   1:  PR[91,1] = PR[90,1] + 5.124;
   1:  PR[91,2] = PR[90,2] + -25.646;
   1:L PR[91] R[100]mm/sec CNT100;
   1:  PR[91,1] = PR[90,1] + 6.998;
   1:  PR[91,2] = PR[90,2] + -25.330;
   1:L PR[91] R[100]mm/sec CNT100;
   1:  PR[91,1] = PR[90,1] + 9.946;
   1:  PR[91,2] = PR[90,2] + -24.476;
   1:L PR[91] R[100]mm/sec CNT100;
   1:  PR[91,1] = PR[90,1] + 11.813;
   1:  PR[91,2] = PR[90,2] + -23.728;
   1:L PR[91] R[100]mm/sec CNT100;
   1:  PR[91,1] = PR[90,1] + 14.404;
   1:  PR[91,2] = PR[90,2] + -22.433;
   1:L PR[91] R[100]mm/sec CNT100;
   1:  PR[91,1] = PR[90,1] + 16.150;
   1:  PR[91,2] = PR[90,2] + -21.252;
   1:L PR[91] R[100]mm/sec CNT100;
   1:  PR[91,1] = PR[90,1] + 18.488;
   1:  PR[91,2] = PR[90,2] + -19.489;
   1:L PR[91] R[100]mm/sec CNT100;
   1:  PR[91,1] = PR[90,1] + 19.988;
   1:  PR[91,2] = PR[90,2] + -17.914;
   1:L PR[91] R[100]mm/sec CNT100;
   1:  PR[91,1] = PR[90,1] + 22.105;
   1:  PR[91,2] = PR[90,2] + -15.542;
   1:L PR[91] R[100]mm/sec CNT100;
   1:  PR[91,1] = PR[90,1] + 23.235;
   1:  PR[91,2] = PR[90,2] + -13.678;
   1:L PR[91] R[100]mm/sec CNT100;
   1:  PR[91,1] = PR[90,1] + 24.761;
   1:  PR[91,2] = PR[90,2] + -11.061;
   1:L PR[91] R[100]mm/sec CNT100;
   1:  PR[91,1] = PR[90,1] + 25.483;
   1:  PR[91,2] = PR[90,2] + -8.945;
   1:L PR[91] R[100]mm/sec CNT100;
   1:  PR[91,1] = PR[90,1] + 26.090;
   1:  PR[91,2] = PR[90,2] + -7.419;
   1:L PR[91] R[100]mm/sec CNT100;
   1:  PR[91,1] = PR[90,1] + 26.501;
   1:  PR[91,2] = PR[90,2] + -5.955;
   1:L PR[91] R[100]mm/sec CNT100;
   1:  PR[91,1] = PR[90,1] + 26.770;
   1:  PR[91,2] = PR[90,2] + -4.345;
   1:L PR[91] R[100]mm/sec CNT100;
   1:  PR[91,1] = PR[90,1] + 27.018;
   1:  PR[91,2] = PR[90,2] + -2.078;
   1:L PR[91] R[100]mm/sec CNT100;
   1:  PR[91,1] = PR[90,1] + 27.107;
   1:  PR[91,2] = PR[90,2] + -0.484;
   1:L PR[91] R[100]mm/sec CNT100;
   1:  PR[91,1] = PR[90,1] + 26.536;
   1:  PR[91,2] = PR[90,2] + 4.905;
   1:L PR[91] R[100]mm/sec CNT100;
   1:  PR[91,1] = PR[90,1] + 25.602;
   1:  PR[91,2] = PR[90,2] + 7.850;
   1:L PR[91] R[100]mm/sec CNT100;
   1:  PR[91,1] = PR[90,1] + 24.902;
   1:  PR[91,2] = PR[90,2] + 9.901;
   1:L PR[91] R[100]mm/sec CNT100;
   1:  PR[91,1] = PR[90,1] + 23.362;
   1:  PR[91,2] = PR[90,2] + 12.656;
   1:L PR[91] R[100]mm/sec CNT100;
   1:  PR[91,1] = PR[90,1] + 22.206;
   1:  PR[91,2] = PR[90,2] + 14.563;
   1:L PR[91] R[100]mm/sec CNT100;
   1:  PR[91,1] = PR[90,1] + 21.245;
   1:  PR[91,2] = PR[90,2] + 15.786;
   1:L PR[91] R[100]mm/sec CNT100;
   1:  PR[91,1] = PR[90,1] + 19.705;
   1:  PR[91,2] = PR[90,2] + 17.404;
   1:L PR[91] R[100]mm/sec CNT100;
   1:  PR[91,1] = PR[90,1] + 18.475;
   1:  PR[91,2] = PR[90,2] + 18.659;
   1:L PR[91] R[100]mm/sec CNT100;
   1:  PR[91,1] = PR[90,1] + 17.022;
   1:  PR[91,2] = PR[90,2] + 19.828;
   1:L PR[91] R[100]mm/sec CNT100;
   1:  PR[91,1] = PR[90,1] + 15.212;
   1:  PR[91,2] = PR[90,2] + 21.053;
   1:L PR[91] R[100]mm/sec CNT100;
   1:  PR[91,1] = PR[90,1] + 13.555;
   1:  PR[91,2] = PR[90,2] + 22.079;
   1:L PR[91] R[100]mm/sec CNT100;
   1:  PR[91,1] = PR[90,1] + 11.797;
   1:  PR[91,2] = PR[90,2] + 22.888;
   1:L PR[91] R[100]mm/sec CNT100;
   1:  PR[91,1] = PR[90,1] + 9.812;
   1:  PR[91,2] = PR[90,2] + 23.683;
   1:L PR[91] R[100]mm/sec CNT100;
   1:  PR[91,1] = PR[90,1] + 7.974;
   1:  PR[91,2] = PR[90,2] + 24.268;
   1:L PR[91] R[100]mm/sec CNT100;
   1:  PR[91,1] = PR[90,1] + 5.960;
   1:  PR[91,2] = PR[90,2] + 24.606;
   1:L PR[91] R[100]mm/sec CNT100;
   1:  PR[91,1] = PR[90,1] + 3.894;
   1:  PR[91,2] = PR[90,2] + 24.993;
   1:L PR[91] R[100]mm/sec CNT100;
   1:  PR[91,1] = PR[90,1] + 1.941;
   1:  PR[91,2] = PR[90,2] + 25.113;
   1:L PR[91] R[100]mm/sec CNT100;
   1:  PR[91,1] = PR[90,1] + -0.146;
   1:  PR[91,2] = PR[90,2] + 25.027;
   1:L PR[91] R[100]mm/sec CNT100;
   1:  PR[91] = PR[90];
   1:  PR[91,1] = PR[90,1] + -1.780;
   1:  PR[91,2] = PR[90,2] + 25.420;
   1:  PR[91,3] = PR[90,3] + 71.695;
   1:L PR[91] R[100]mm/sec CNT100;
   1:  PR[91,1] = PR[90,1] + -4.146;
   1:  PR[91,2] = PR[90,2] + 25.274;
   1:L PR[91] R[100]mm/sec CNT100;
   1:  PR[91,1] = PR[90,1] + -5.565;
   1:  PR[91,2] = PR[90,2] + 25.035;
   1:L PR[91] R[100]mm/sec CNT100;
   1:  PR[91,1] = PR[90,1] + -7.940;
   1:  PR[91,2] = PR[90,2] + 24.591;
   1:L PR[91] R[100]mm/sec CNT100;
   1:  PR[91,1] = PR[90,1] + -10.180;
   1:  PR[91,2] = PR[90,2] + 23.878;
   1:L PR[91] R[100]mm/sec CNT100;
   1:  PR[91,1] = PR[90,1] + -11.552;
   1:  PR[91,2] = PR[90,2] + 23.329;
   1:L PR[91] R[100]mm/sec CNT100;
   1:  PR[91,1] = PR[90,1] + -13.642;
   1:  PR[91,2] = PR[90,2] + 22.367;
   1:L PR[91] R[100]mm/sec CNT100;
   1:  PR[91,1] = PR[90,1] + -14.917;
   1:  PR[91,2] = PR[90,2] + 21.506;
   1:L PR[91] R[100]mm/sec CNT100;
   1:  PR[91,1] = PR[90,1] + -16.981;
   1:  PR[91,2] = PR[90,2] + 20.227;
   1:L PR[91] R[100]mm/sec CNT100;
   1:  PR[91,1] = PR[90,1] + -18.712;
   1:  PR[91,2] = PR[90,2] + 18.833;
   1:L PR[91] R[100]mm/sec CNT100;
   1:  PR[91,1] = PR[90,1] + -19.758;
   1:  PR[91,2] = PR[90,2] + 17.736;
   1:L PR[91] R[100]mm/sec CNT100;
   1:  PR[91,1] = PR[90,1] + -22.355;
   1:  PR[91,2] = PR[90,2] + 14.827;
   1:L PR[91] R[100]mm/sec CNT100;
   1:  PR[91,1] = PR[90,1] + -23.115;
   1:  PR[91,2] = PR[90,2] + 13.573;
   1:L PR[91] R[100]mm/sec CNT100;
   1:  PR[91,1] = PR[90,1] + -24.999;
   1:  PR[91,2] = PR[90,2] + 10.343;
   1:L PR[91] R[100]mm/sec CNT100;
   1:  PR[91,1] = PR[90,1] + -25.488;
   1:  PR[91,2] = PR[90,2] + 8.909;
   1:L PR[91] R[100]mm/sec CNT100;
   1:  PR[91,1] = PR[90,1] + -26.233;
   1:  PR[91,2] = PR[90,2] + 7.034;
   1:L PR[91] R[100]mm/sec CNT100;
   1:  PR[91,1] = PR[90,1] + -26.751;
   1:  PR[91,2] = PR[90,2] + 5.192;
   1:L PR[91] R[100]mm/sec CNT100;
   1:  PR[91,1] = PR[90,1] + -27.087;
   1:  PR[91,2] = PR[90,2] + 3.184;
   1:L PR[91] R[100]mm/sec CNT100;
   1:  PR[91,1] = PR[90,1] + -27.255;
   1:  PR[91,2] = PR[90,2] + 1.644;
   1:L PR[91] R[100]mm/sec CNT100;
   1:  PR[91,1] = PR[90,1] + -27.367;
   1:  PR[91,2] = PR[90,2] + -0.364;
   1:L PR[91] R[100]mm/sec CNT100;
   1:  PR[91,1] = PR[90,1] + -26.796;
   1:  PR[91,2] = PR[90,2] + -5.788;
   1:L PR[91] R[100]mm/sec CNT100;
   1:  PR[91,1] = PR[90,1] + -25.639;
   1:  PR[91,2] = PR[90,2] + -9.436;
   1:L PR[91] R[100]mm/sec CNT100;
   1:  PR[91,1] = PR[90,1] + -25.172;
   1:  PR[91,2] = PR[90,2] + -10.805;
   1:L PR[91] R[100]mm/sec CNT100;
   1:  PR[91,1] = PR[90,1] + -23.273;
   1:  PR[91,2] = PR[90,2] + -14.201;
   1:L PR[91] R[100]mm/sec CNT100;
   1:  PR[91,1] = PR[90,1] + -22.487;
   1:  PR[91,2] = PR[90,2] + -15.498;
   1:L PR[91] R[100]mm/sec CNT100;
   1:  PR[91,1] = PR[90,1] + -21.291;
   1:  PR[91,2] = PR[90,2] + -17.021;
   1:L PR[91] R[100]mm/sec CNT100;
   1:  PR[91,1] = PR[90,1] + -20.228;
   1:  PR[91,2] = PR[90,2] + -18.137;
   1:L PR[91] R[100]mm/sec CNT100;
   1:  PR[91,1] = PR[90,1] + -18.757;
   1:  PR[91,2] = PR[90,2] + -19.638;
   1:L PR[91] R[100]mm/sec CNT100;
   1:  PR[91,1] = PR[90,1] + -15.723;
   1:  PR[91,2] = PR[90,2] + -21.903;
   1:L PR[91] R[100]mm/sec CNT100;
   1:  PR[91,1] = PR[90,1] + -14.553;
   1:  PR[91,2] = PR[90,2] + -22.694;
   1:L PR[91] R[100]mm/sec CNT100;
   1:  PR[91,1] = PR[90,1] + -11.293;
   1:  PR[91,2] = PR[90,2] + -24.274;
   1:L PR[91] R[100]mm/sec CNT100;
   1:  PR[91,1] = PR[90,1] + -10.048;
   1:  PR[91,2] = PR[90,2] + -24.773;
   1:L PR[91] R[100]mm/sec CNT100;
   1:  PR[91,1] = PR[90,1] + -6.562;
   1:  PR[91,2] = PR[90,2] + -25.731;
   1:L PR[91] R[100]mm/sec CNT100;
   1:  PR[91,1] = PR[90,1] + -5.323;
   1:  PR[91,2] = PR[90,2] + -25.940;
   1:L PR[91] R[100]mm/sec CNT100;
   1:  PR[91,1] = PR[90,1] + -1.628;
   1:  PR[91,2] = PR[90,2] + -26.261;
   1:L PR[91] R[100]mm/sec CNT100;
   1:  PR[91,1] = PR[90,1] + -0.309;
   1:  PR[91,2] = PR[90,2] + -26.206;
   1:L PR[91] R[100]mm/sec CNT100;
   1:  PR[91,1] = PR[90,1] + 1.137;
   1:  PR[91,2] = PR[90,2] + -26.261;
   1:L PR[91] R[100]mm/sec CNT100;
   1:  PR[91,1] = PR[90,1] + 5.091;
   1:  PR[91,2] = PR[90,2] + -25.894;
   1:L PR[91] R[100]mm/sec CNT100;
   1:  PR[91,1] = PR[90,1] + 6.320;
   1:  PR[91,2] = PR[90,2] + -25.686;
   1:L PR[91] R[100]mm/sec CNT100;
   1:  PR[91,1] = PR[90,1] + 9.853;
   1:  PR[91,2] = PR[90,2] + -24.664;
   1:L PR[91] R[100]mm/sec CNT100;
   1:  PR[91,1] = PR[90,1] + 11.098;
   1:  PR[91,2] = PR[90,2] + -24.165;
   1:L PR[91] R[100]mm/sec CNT100;
   1:  PR[91,1] = PR[90,1] + 14.232;
   1:  PR[91,2] = PR[90,2] + -22.598;
   1:L PR[91] R[100]mm/sec CNT100;
   1:  PR[91,1] = PR[90,1] + 15.409;
   1:  PR[91,2] = PR[90,2] + -21.802;
   1:L PR[91] R[100]mm/sec CNT100;
   1:  PR[91,1] = PR[90,1] + 18.260;
   1:  PR[91,2] = PR[90,2] + -19.652;
   1:L PR[91] R[100]mm/sec CNT100;
   1:  PR[91,1] = PR[90,1] + 19.279;
   1:  PR[91,2] = PR[90,2] + -18.582;
   1:L PR[91] R[100]mm/sec CNT100;
   1:  PR[91,1] = PR[90,1] + 21.876;
   1:  PR[91,2] = PR[90,2] + -15.672;
   1:L PR[91] R[100]mm/sec CNT100;
   1:  PR[91,1] = PR[90,1] + 22.636;
   1:  PR[91,2] = PR[90,2] + -14.418;
   1:L PR[91] R[100]mm/sec CNT100;
   1:  PR[91,1] = PR[90,1] + 24.520;
   1:  PR[91,2] = PR[90,2] + -11.188;
   1:L PR[91] R[100]mm/sec CNT100;
   1:  PR[91,1] = PR[90,1] + 25.009;
   1:  PR[91,2] = PR[90,2] + -9.755;
   1:L PR[91] R[100]mm/sec CNT100;
   1:  PR[91,1] = PR[90,1] + 25.754;
   1:  PR[91,2] = PR[90,2] + -7.880;
   1:L PR[91] R[100]mm/sec CNT100;
   1:  PR[91,1] = PR[90,1] + 26.271;
   1:  PR[91,2] = PR[90,2] + -6.039;
   1:L PR[91] R[100]mm/sec CNT100;
   1:  PR[91,1] = PR[90,1] + 26.607;
   1:  PR[91,2] = PR[90,2] + -4.032;
   1:L PR[91] R[100]mm/sec CNT100;
   1:  PR[91,1] = PR[90,1] + 26.776;
   1:  PR[91,2] = PR[90,2] + -2.491;
   1:L PR[91] R[100]mm/sec CNT100;
   1:  PR[91,1] = PR[90,1] + 26.887;
   1:  PR[91,2] = PR[90,2] + -0.483;
   1:L PR[91] R[100]mm/sec CNT100;
   1:  PR[91,1] = PR[90,1] + 26.317;
   1:  PR[91,2] = PR[90,2] + 4.939;
   1:L PR[91] R[100]mm/sec CNT100;
   1:  PR[91,1] = PR[90,1] + 25.160;
   1:  PR[91,2] = PR[90,2] + 8.588;
   1:L PR[91] R[100]mm/sec CNT100;
   1:  PR[91,1] = PR[90,1] + 24.693;
   1:  PR[91,2] = PR[90,2] + 9.956;
   1:L PR[91] R[100]mm/sec CNT100;
   1:  PR[91,1] = PR[90,1] + 22.793;
   1:  PR[91,2] = PR[90,2] + 13.354;
   1:L PR[91] R[100]mm/sec CNT100;
   1:  PR[91,1] = PR[90,1] + 22.006;
   1:  PR[91,2] = PR[90,2] + 14.652;
   1:L PR[91] R[100]mm/sec CNT100;
   1:  PR[91,1] = PR[90,1] + 20.811;
   1:  PR[91,2] = PR[90,2] + 16.174;
   1:L PR[91] R[100]mm/sec CNT100;
   1:  PR[91,1] = PR[90,1] + 19.747;
   1:  PR[91,2] = PR[90,2] + 17.291;
   1:L PR[91] R[100]mm/sec CNT100;
   1:  PR[91,1] = PR[90,1] + 18.247;
   1:  PR[91,2] = PR[90,2] + 18.822;
   1:L PR[91] R[100]mm/sec CNT100;
   1:  PR[91,1] = PR[90,1] + 16.464;
   1:  PR[91,2] = PR[90,2] + 20.257;
   1:L PR[91] R[100]mm/sec CNT100;
   1:  PR[91,1] = PR[90,1] + 15.212;
   1:  PR[91,2] = PR[90,2] + 21.104;
   1:L PR[91] R[100]mm/sec CNT100;
   1:  PR[91,1] = PR[90,1] + 13.205;
   1:  PR[91,2] = PR[90,2] + 22.347;
   1:L PR[91] R[100]mm/sec CNT100;
   1:  PR[91,1] = PR[90,1] + 11.072;
   1:  PR[91,2] = PR[90,2] + 23.329;
   1:L PR[91] R[100]mm/sec CNT100;
   1:  PR[91,1] = PR[90,1] + 9.701;
   1:  PR[91,2] = PR[90,2] + 23.878;
   1:L PR[91] R[100]mm/sec CNT100;
   1:  PR[91,1] = PR[90,1] + 7.481;
   1:  PR[91,2] = PR[90,2] + 24.584;
   1:L PR[91] R[100]mm/sec CNT100;
   1:  PR[91,1] = PR[90,1] + 6.092;
   1:  PR[91,2] = PR[90,2] + 24.818;
   1:L PR[91] R[100]mm/sec CNT100;
   1:  PR[91,1] = PR[90,1] + 3.644;
   1:  PR[91,2] = PR[90,2] + 25.275;
   1:L PR[91] R[100]mm/sec CNT100;
   1:  PR[91,1] = PR[90,1] + 1.303;
   1:  PR[91,2] = PR[90,2] + 25.420;
   1:L PR[91] R[100]mm/sec CNT100;
   1:  PR[91,1] = PR[90,1] + -0.172;
   1:  PR[91,2] = PR[90,2] + 25.359;
   1:L PR[91] R[100]mm/sec CNT100;
   1:  PR[91] = PR[90];
   1:  PR[91,1] = PR[90,1] + -1.142;
   1:  PR[91,2] = PR[90,2] + 25.727;
   1:  PR[91,3] = PR[90,3] + 72.995;
   1:L PR[91] R[100]mm/sec CNT100;
   1:  PR[91,1] = PR[90,1] + -3.897;
   1:  PR[91,2] = PR[90,2] + 25.556;
   1:L PR[91] R[100]mm/sec CNT100;
   1:  PR[91,1] = PR[90,1] + -4.679;
   1:  PR[91,2] = PR[90,2] + 25.425;
   1:L PR[91] R[100]mm/sec CNT100;
   1:  PR[91,1] = PR[90,1] + -7.448;
   1:  PR[91,2] = PR[90,2] + 24.907;
   1:L PR[91] R[100]mm/sec CNT100;
   1:  PR[91,1] = PR[90,1] + -10.070;
   1:  PR[91,2] = PR[90,2] + 24.073;
   1:L PR[91] R[100]mm/sec CNT100;
   1:  PR[91,1] = PR[90,1] + -10.827;
   1:  PR[91,2] = PR[90,2] + 23.769;
   1:L PR[91] R[100]mm/sec CNT100;
   1:  PR[91,1] = PR[90,1] + -13.292;
   1:  PR[91,2] = PR[90,2] + 22.635;
   1:L PR[91] R[100]mm/sec CNT100;
   1:  PR[91,1] = PR[90,1] + -13.998;
   1:  PR[91,2] = PR[90,2] + 22.158;
   1:L PR[91] R[100]mm/sec CNT100;
   1:  PR[91,1] = PR[90,1] + -16.423;
   1:  PR[91,2] = PR[90,2] + 20.656;
   1:L PR[91] R[100]mm/sec CNT100;
   1:  PR[91,1] = PR[90,1] + -18.484;
   1:  PR[91,2] = PR[90,2] + 18.996;
   1:L PR[91] R[100]mm/sec CNT100;
   1:  PR[91,1] = PR[90,1] + -19.049;
   1:  PR[91,2] = PR[90,2] + 18.404;
   1:L PR[91] R[100]mm/sec CNT100;
   1:  PR[91,1] = PR[90,1] + -22.125;
   1:  PR[91,2] = PR[90,2] + 14.957;
   1:L PR[91] R[100]mm/sec CNT100;
   1:  PR[91,1] = PR[90,1] + -22.516;
   1:  PR[91,2] = PR[90,2] + 14.313;
   1:L PR[91] R[100]mm/sec CNT100;
   1:  PR[91,1] = PR[90,1] + -24.757;
   1:  PR[91,2] = PR[90,2] + 10.470;
   1:L PR[91] R[100]mm/sec CNT100;
   1:  PR[91,1] = PR[90,1] + -25.013;
   1:  PR[91,2] = PR[90,2] + 9.720;
   1:L PR[91] R[100]mm/sec CNT100;
   1:  PR[91,1] = PR[90,1] + -25.898;
   1:  PR[91,2] = PR[90,2] + 7.495;
   1:L PR[91] R[100]mm/sec CNT100;
   1:  PR[91,1] = PR[90,1] + -26.521;
   1:  PR[91,2] = PR[90,2] + 5.276;
   1:L PR[91] R[100]mm/sec CNT100;
   1:  PR[91,1] = PR[90,1] + -26.923;
   1:  PR[91,2] = PR[90,2] + 2.871;
   1:L PR[91] R[100]mm/sec CNT100;
   1:  PR[91,1] = PR[90,1] + -27.013;
   1:  PR[91,2] = PR[90,2] + 2.056;
   1:L PR[91] R[100]mm/sec CNT100;
   1:  PR[91,1] = PR[90,1] + -27.147;
   1:  PR[91,2] = PR[90,2] + -0.365;
   1:L PR[91] R[100]mm/sec CNT100;
   1:  PR[91,1] = PR[90,1] + -26.577;
   1:  PR[91,2] = PR[90,2] + -5.823;
   1:L PR[91] R[100]mm/sec CNT100;
   1:  PR[91,1] = PR[90,1] + -25.197;
   1:  PR[91,2] = PR[90,2] + -10.174;
   1:L PR[91] R[100]mm/sec CNT100;
   1:  PR[91,1] = PR[90,1] + -24.963;
   1:  PR[91,2] = PR[90,2] + -10.860;
   1:L PR[91] R[100]mm/sec CNT100;
   1:  PR[91,1] = PR[90,1] + -22.704;
   1:  PR[91,2] = PR[90,2] + -14.899;
   1:L PR[91] R[100]mm/sec CNT100;
   1:  PR[91,1] = PR[90,1] + -22.287;
   1:  PR[91,2] = PR[90,2] + -15.587;
   1:L PR[91] R[100]mm/sec CNT100;
   1:  PR[91,1] = PR[90,1] + -20.857;
   1:  PR[91,2] = PR[90,2] + -17.409;
   1:L PR[91] R[100]mm/sec CNT100;
   1:  PR[91,1] = PR[90,1] + -20.271;
   1:  PR[91,2] = PR[90,2] + -18.024;
   1:L PR[91] R[100]mm/sec CNT100;
   1:  PR[91,1] = PR[90,1] + -18.529;
   1:  PR[91,2] = PR[90,2] + -19.802;
   1:L PR[91] R[100]mm/sec CNT100;
   1:  PR[91,1] = PR[90,1] + -14.954;
   1:  PR[91,2] = PR[90,2] + -22.470;
   1:L PR[91] R[100]mm/sec CNT100;
   1:  PR[91,1] = PR[90,1] + -14.353;
   1:  PR[91,2] = PR[90,2] + -22.876;
   1:L PR[91] R[100]mm/sec CNT100;
   1:  PR[91,1] = PR[90,1] + -10.529;
   1:  PR[91,2] = PR[90,2] + -24.729;
   1:L PR[91] R[100]mm/sec CNT100;
   1:  PR[91,1] = PR[90,1] + -9.910;
   1:  PR[91,2] = PR[90,2] + -24.978;
   1:L PR[91] R[100]mm/sec CNT100;
   1:  PR[91,1] = PR[90,1] + -5.845;
   1:  PR[91,2] = PR[90,2] + -26.095;
   1:L PR[91] R[100]mm/sec CNT100;
   1:  PR[91,1] = PR[90,1] + -5.252;
   1:  PR[91,2] = PR[90,2] + -26.195;
   1:L PR[91] R[100]mm/sec CNT100;
   1:  PR[91,1] = PR[90,1] + -0.972;
   1:  PR[91,2] = PR[90,2] + -26.566;
   1:L PR[91] R[100]mm/sec CNT100;
   1:  PR[91,1] = PR[90,1] + -0.283;
   1:  PR[91,2] = PR[90,2] + -26.538;
   1:L PR[91] R[100]mm/sec CNT100;
   1:  PR[91,1] = PR[90,1] + 0.480;
   1:  PR[91,2] = PR[90,2] + -26.567;
   1:L PR[91] R[100]mm/sec CNT100;
   1:  PR[91,1] = PR[90,1] + 5.058;
   1:  PR[91,2] = PR[90,2] + -26.142;
   1:L PR[91] R[100]mm/sec CNT100;
   1:  PR[91,1] = PR[90,1] + 5.643;
   1:  PR[91,2] = PR[90,2] + -26.043;
   1:L PR[91] R[100]mm/sec CNT100;
   1:  PR[91,1] = PR[90,1] + 9.761;
   1:  PR[91,2] = PR[90,2] + -24.851;
   1:L PR[91] R[100]mm/sec CNT100;
   1:  PR[91,1] = PR[90,1] + 10.383;
   1:  PR[91,2] = PR[90,2] + -24.602;
   1:L PR[91] R[100]mm/sec CNT100;
   1:  PR[91,1] = PR[90,1] + 14.059;
   1:  PR[91,2] = PR[90,2] + -22.764;
   1:L PR[91] R[100]mm/sec CNT100;
   1:  PR[91,1] = PR[90,1] + 14.669;
   1:  PR[91,2] = PR[90,2] + -22.351;
   1:L PR[91] R[100]mm/sec CNT100;
   1:  PR[91,1] = PR[90,1] + 18.032;
   1:  PR[91,2] = PR[90,2] + -19.816;
   1:L PR[91] R[100]mm/sec CNT100;
   1:  PR[91,1] = PR[90,1] + 18.570;
   1:  PR[91,2] = PR[90,2] + -19.250;
   1:L PR[91] R[100]mm/sec CNT100;
   1:  PR[91,1] = PR[90,1] + 21.647;
   1:  PR[91,2] = PR[90,2] + -15.803;
   1:L PR[91] R[100]mm/sec CNT100;
   1:  PR[91,1] = PR[90,1] + 22.037;
   1:  PR[91,2] = PR[90,2] + -15.159;
   1:L PR[91] R[100]mm/sec CNT100;
   1:  PR[91,1] = PR[90,1] + 24.279;
   1:  PR[91,2] = PR[90,2] + -11.315;
   1:L PR[91] R[100]mm/sec CNT100;
   1:  PR[91,1] = PR[90,1] + 24.534;
   1:  PR[91,2] = PR[90,2] + -10.566;
   1:L PR[91] R[100]mm/sec CNT100;
   1:  PR[91,1] = PR[90,1] + 25.419;
   1:  PR[91,2] = PR[90,2] + -8.341;
   1:L PR[91] R[100]mm/sec CNT100;
   1:  PR[91,1] = PR[90,1] + 26.041;
   1:  PR[91,2] = PR[90,2] + -6.123;
   1:L PR[91] R[100]mm/sec CNT100;
   1:  PR[91,1] = PR[90,1] + 26.444;
   1:  PR[91,2] = PR[90,2] + -3.718;
   1:L PR[91] R[100]mm/sec CNT100;
   1:  PR[91,1] = PR[90,1] + 26.533;
   1:  PR[91,2] = PR[90,2] + -2.903;
   1:L PR[91] R[100]mm/sec CNT100;
   1:  PR[91,1] = PR[90,1] + 26.668;
   1:  PR[91,2] = PR[90,2] + -0.482;
   1:L PR[91] R[100]mm/sec CNT100;
   1:  PR[91,1] = PR[90,1] + 26.098;
   1:  PR[91,2] = PR[90,2] + 4.972;
   1:L PR[91] R[100]mm/sec CNT100;
   1:  PR[91,1] = PR[90,1] + 24.718;
   1:  PR[91,2] = PR[90,2] + 9.326;
   1:L PR[91] R[100]mm/sec CNT100;
   1:  PR[91,1] = PR[90,1] + 24.484;
   1:  PR[91,2] = PR[90,2] + 10.011;
   1:L PR[91] R[100]mm/sec CNT100;
   1:  PR[91,1] = PR[90,1] + 22.223;
   1:  PR[91,2] = PR[90,2] + 14.053;
   1:L PR[91] R[100]mm/sec CNT100;
   1:  PR[91,1] = PR[90,1] + 21.807;
   1:  PR[91,2] = PR[90,2] + 14.741;
   1:L PR[91] R[100]mm/sec CNT100;
   1:  PR[91,1] = PR[90,1] + 20.376;
   1:  PR[91,2] = PR[90,2] + 16.562;
   1:L PR[91] R[100]mm/sec CNT100;
   1:  PR[91,1] = PR[90,1] + 19.789;
   1:  PR[91,2] = PR[90,2] + 17.179;
   1:L PR[91] R[100]mm/sec CNT100;
   1:  PR[91,1] = PR[90,1] + 18.019;
   1:  PR[91,2] = PR[90,2] + 18.985;
   1:L PR[91] R[100]mm/sec CNT100;
   1:  PR[91,1] = PR[90,1] + 15.906;
   1:  PR[91,2] = PR[90,2] + 20.686;
   1:L PR[91] R[100]mm/sec CNT100;
   1:  PR[91,1] = PR[90,1] + 15.213;
   1:  PR[91,2] = PR[90,2] + 21.155;
   1:L PR[91] R[100]mm/sec CNT100;
   1:  PR[91,1] = PR[90,1] + 12.855;
   1:  PR[91,2] = PR[90,2] + 22.615;
   1:L PR[91] R[100]mm/sec CNT100;
   1:  PR[91,1] = PR[90,1] + 10.347;
   1:  PR[91,2] = PR[90,2] + 23.769;
   1:L PR[91] R[100]mm/sec CNT100;
   1:  PR[91,1] = PR[90,1] + 9.590;
   1:  PR[91,2] = PR[90,2] + 24.073;
   1:L PR[91] R[100]mm/sec CNT100;
   1:  PR[91,1] = PR[90,1] + 6.988;
   1:  PR[91,2] = PR[90,2] + 24.900;
   1:L PR[91] R[100]mm/sec CNT100;
   1:  PR[91,1] = PR[90,1] + 6.224;
   1:  PR[91,2] = PR[90,2] + 25.029;
   1:L PR[91] R[100]mm/sec CNT100;
   1:  PR[91,1] = PR[90,1] + 3.394;
   1:  PR[91,2] = PR[90,2] + 25.558;
   1:L PR[91] R[100]mm/sec CNT100;
   1:  PR[91,1] = PR[90,1] + 0.665;
   1:  PR[91,2] = PR[90,2] + 25.726;
   1:L PR[91] R[100]mm/sec CNT100;
   1:  PR[91,1] = PR[90,1] + -0.199;
   1:  PR[91,2] = PR[90,2] + 25.691;
   1:L PR[91] R[100]mm/sec CNT100;
   1:  PR[91] = PR[90];
   1:  PR[91,1] = PR[90,1] + -0.504;
   1:  PR[91,2] = PR[90,2] + 26.033;
   1:  PR[91,3] = PR[90,3] + 74.295;
   1:L PR[91] R[100]mm/sec CNT100;
   1:  PR[91,1] = PR[90,1] + -3.627;
   1:  PR[91,2] = PR[90,2] + 25.840;
   1:L PR[91] R[100]mm/sec CNT100;
   1:  PR[91,1] = PR[90,1] + -6.957;
   1:  PR[91,2] = PR[90,2] + 25.223;
   1:L PR[91] R[100]mm/sec CNT100;
   1:  PR[91,1] = PR[90,1] + -9.959;
   1:  PR[91,2] = PR[90,2] + 24.267;
   1:L PR[91] R[100]mm/sec CNT100;
   1:  PR[91,1] = PR[90,1] + -10.102;
   1:  PR[91,2] = PR[90,2] + 24.210;
   1:L PR[91] R[100]mm/sec CNT100;
   1:  PR[91,1] = PR[90,1] + -12.942;
   1:  PR[91,2] = PR[90,2] + 22.903;
   1:L PR[91] R[100]mm/sec CNT100;
   1:  PR[91,1] = PR[90,1] + -13.079;
   1:  PR[91,2] = PR[90,2] + 22.810;
   1:L PR[91] R[100]mm/sec CNT100;
   1:  PR[91,1] = PR[90,1] + -15.865;
   1:  PR[91,2] = PR[90,2] + 21.085;
   1:L PR[91] R[100]mm/sec CNT100;
   1:  PR[91,1] = PR[90,1] + -18.227;
   1:  PR[91,2] = PR[90,2] + 19.183;
   1:L PR[91] R[100]mm/sec CNT100;
   1:  PR[91,1] = PR[90,1] + -21.884;
   1:  PR[91,2] = PR[90,2] + 15.100;
   1:L PR[91] R[100]mm/sec CNT100;
   1:  PR[91,1] = PR[90,1] + -24.516;
   1:  PR[91,2] = PR[90,2] + 10.596;
   1:L PR[91] R[100]mm/sec CNT100;
   1:  PR[91,1] = PR[90,1] + -24.538;
   1:  PR[91,2] = PR[90,2] + 10.531;
   1:L PR[91] R[100]mm/sec CNT100;
   1:  PR[91,1] = PR[90,1] + -25.562;
   1:  PR[91,2] = PR[90,2] + 7.957;
   1:L PR[91] R[100]mm/sec CNT100;
   1:  PR[91,1] = PR[90,1] + -26.291;
   1:  PR[91,2] = PR[90,2] + 5.361;
   1:L PR[91] R[100]mm/sec CNT100;
   1:  PR[91,1] = PR[90,1] + -26.760;
   1:  PR[91,2] = PR[90,2] + 2.559;
   1:L PR[91] R[100]mm/sec CNT100;
   1:  PR[91,1] = PR[90,1] + -26.770;
   1:  PR[91,2] = PR[90,2] + 2.469;
   1:L PR[91] R[100]mm/sec CNT100;
   1:  PR[91,1] = PR[90,1] + -26.928;
   1:  PR[91,2] = PR[90,2] + -0.366;
   1:L PR[91] R[100]mm/sec CNT100;
   1:  PR[91,1] = PR[90,1] + -26.358;
   1:  PR[91,2] = PR[90,2] + -5.856;
   1:L PR[91] R[100]mm/sec CNT100;
   1:  PR[91,1] = PR[90,1] + -24.741;
   1:  PR[91,2] = PR[90,2] + -10.937;
   1:L PR[91] R[100]mm/sec CNT100;
   1:  PR[91,1] = PR[90,1] + -22.135;
   1:  PR[91,2] = PR[90,2] + -15.598;
   1:L PR[91] R[100]mm/sec CNT100;
   1:  PR[91,1] = PR[90,1] + -22.088;
   1:  PR[91,2] = PR[90,2] + -15.676;
   1:L PR[91] R[100]mm/sec CNT100;
   1:  PR[91,1] = PR[90,1] + -20.432;
   1:  PR[91,2] = PR[90,2] + -17.784;
   1:L PR[91] R[100]mm/sec CNT100;
   1:  PR[91,1] = PR[90,1] + -18.299;
   1:  PR[91,2] = PR[90,2] + -19.966;
   1:L PR[91] R[100]mm/sec CNT100;
   1:  PR[91,1] = PR[90,1] + -14.185;
   1:  PR[91,2] = PR[90,2] + -23.037;
   1:L PR[91] R[100]mm/sec CNT100;
   1:  PR[91,1] = PR[90,1] + -14.153;
   1:  PR[91,2] = PR[90,2] + -23.058;
   1:L PR[91] R[100]mm/sec CNT100;
   1:  PR[91,1] = PR[90,1] + -9.769;
   1:  PR[91,2] = PR[90,2] + -25.183;
   1:L PR[91] R[100]mm/sec CNT100;
   1:  PR[91,1] = PR[90,1] + -5.151;
   1:  PR[91,2] = PR[90,2] + -26.452;
   1:L PR[91] R[100]mm/sec CNT100;
   1:  PR[91,1] = PR[90,1] + -0.265;
   1:  PR[91,2] = PR[90,2] + -26.877;
   1:L PR[91] R[100]mm/sec CNT100;
   1:  PR[91,1] = PR[90,1] + -0.222;
   1:L PR[91] R[100]mm/sec CNT100;
   1:  PR[91,1] = PR[90,1] + 4.988;
   1:  PR[91,2] = PR[90,2] + -26.393;
   1:L PR[91] R[100]mm/sec CNT100;
   1:  PR[91,1] = PR[90,1] + 9.668;
   1:  PR[91,2] = PR[90,2] + -25.038;
   1:L PR[91] R[100]mm/sec CNT100;
   1:  PR[91,1] = PR[90,1] + 13.887;
   1:  PR[91,2] = PR[90,2] + -22.929;
   1:L PR[91] R[100]mm/sec CNT100;
   1:  PR[91,1] = PR[90,1] + 13.928;
   1:  PR[91,2] = PR[90,2] + -22.901;
   1:L PR[91] R[100]mm/sec CNT100;
   1:  PR[91,1] = PR[90,1] + 17.774;
   1:  PR[91,2] = PR[90,2] + -20.001;
   1:L PR[91] R[100]mm/sec CNT100;
   1:  PR[91,1] = PR[90,1] + 21.405;
   1:  PR[91,2] = PR[90,2] + -15.946;
   1:L PR[91] R[100]mm/sec CNT100;
   1:  PR[91,1] = PR[90,1] + 24.038;
   1:  PR[91,2] = PR[90,2] + -11.441;
   1:L PR[91] R[100]mm/sec CNT100;
   1:  PR[91,1] = PR[90,1] + 24.060;
   1:  PR[91,2] = PR[90,2] + -11.376;
   1:L PR[91] R[100]mm/sec CNT100;
   1:  PR[91,1] = PR[90,1] + 25.083;
   1:  PR[91,2] = PR[90,2] + -8.802;
   1:L PR[91] R[100]mm/sec CNT100;
   1:  PR[91,1] = PR[90,1] + 25.811;
   1:  PR[91,2] = PR[90,2] + -6.207;
   1:L PR[91] R[100]mm/sec CNT100;
   1:  PR[91,1] = PR[90,1] + 26.280;
   1:  PR[91,2] = PR[90,2] + -3.405;
   1:L PR[91] R[100]mm/sec CNT100;
   1:  PR[91,1] = PR[90,1] + 26.290;
   1:  PR[91,2] = PR[90,2] + -3.316;
   1:L PR[91] R[100]mm/sec CNT100;
   1:  PR[91,1] = PR[90,1] + 26.448;
   1:  PR[91,2] = PR[90,2] + -0.481;
   1:L PR[91] R[100]mm/sec CNT100;
   1:  PR[91,1] = PR[90,1] + 25.879;
   1:  PR[91,2] = PR[90,2] + 5.005;
   1:L PR[91] R[100]mm/sec CNT100;
   1:  PR[91,1] = PR[90,1] + 24.263;
   1:  PR[91,2] = PR[90,2] + 10.086;
   1:L PR[91] R[100]mm/sec CNT100;
   1:  PR[91,1] = PR[90,1] + 21.582;
   1:  PR[91,2] = PR[90,2] + 14.861;
   1:L PR[91] R[100]mm/sec CNT100;
   1:  PR[91,1] = PR[90,1] + 19.951;
   1:  PR[91,2] = PR[90,2] + 16.938;
   1:L PR[91] R[100]mm/sec CNT100;
   1:  PR[91,1] = PR[90,1] + 17.790;
   1:  PR[91,2] = PR[90,2] + 19.149;
   1:L PR[91] R[100]mm/sec CNT100;
   1:  PR[91,1] = PR[90,1] + 15.348;
   1:  PR[91,2] = PR[90,2] + 21.115;
   1:L PR[91] R[100]mm/sec CNT100;
   1:  PR[91,1] = PR[90,1] + 15.214;
   1:  PR[91,2] = PR[90,2] + 21.205;
   1:L PR[91] R[100]mm/sec CNT100;
   1:  PR[91,1] = PR[90,1] + 12.505;
   1:  PR[91,2] = PR[90,2] + 22.883;
   1:L PR[91] R[100]mm/sec CNT100;
   1:  PR[91,1] = PR[90,1] + 9.622;
   1:  PR[91,2] = PR[90,2] + 24.210;
   1:L PR[91] R[100]mm/sec CNT100;
   1:  PR[91,1] = PR[90,1] + 9.479;
   1:  PR[91,2] = PR[90,2] + 24.267;
   1:L PR[91] R[100]mm/sec CNT100;
   1:  PR[91,1] = PR[90,1] + 6.476;
   1:  PR[91,2] = PR[90,2] + 25.223;
   1:L PR[91] R[100]mm/sec CNT100;
   1:  PR[91,1] = PR[90,1] + 3.145;
   1:  PR[91,2] = PR[90,2] + 25.841;
   1:L PR[91] R[100]mm/sec CNT100;
   1:  PR[91,1] = PR[90,1] + 0.026;
   1:  PR[91,2] = PR[90,2] + 26.033;
   1:L PR[91] R[100]mm/sec CNT100;
   1:  PR[91,1] = PR[90,1] + -0.225;
   1:  PR[91,2] = PR[90,2] + 26.023;
   1:L PR[91] R[100]mm/sec CNT100;
   1:  PR[91] = PR[90];
   1:  PR[91,1] = PR[90,1] + -0.592;
   1:  PR[91,2] = PR[90,2] + 26.151;
   1:  PR[91,3] = PR[90,3] + 75.595;
   1:L PR[91] R[100]mm/sec CNT100;
   1:  PR[91,1] = PR[90,1] + -3.502;
   1:  PR[91,2] = PR[90,2] + 25.971;
   1:L PR[91] R[100]mm/sec CNT100;
   1:  PR[91,1] = PR[90,1] + -6.373;
   1:  PR[91,2] = PR[90,2] + 25.434;
   1:L PR[91] R[100]mm/sec CNT100;
   1:  PR[91,1] = PR[90,1] + -7.054;
   1:  PR[91,2] = PR[90,2] + 25.266;
   1:L PR[91] R[100]mm/sec CNT100;
   1:  PR[91,1] = PR[90,1] + -9.826;
   1:  PR[91,2] = PR[90,2] + 24.384;
   1:L PR[91] R[100]mm/sec CNT100;
   1:  PR[91,1] = PR[90,1] + -12.484;
   1:  PR[91,2] = PR[90,2] + 23.160;
   1:L PR[91] R[100]mm/sec CNT100;
   1:  PR[91,1] = PR[90,1] + -13.106;
   1:  PR[91,2] = PR[90,2] + 22.834;
   1:L PR[91] R[100]mm/sec CNT100;
   1:  PR[91,1] = PR[90,1] + -15.575;
   1:  PR[91,2] = PR[90,2] + 21.305;
   1:L PR[91] R[100]mm/sec CNT100;
   1:  PR[91,1] = PR[90,1] + -17.858;
   1:  PR[91,2] = PR[90,2] + 19.467;
   1:L PR[91] R[100]mm/sec CNT100;
   1:  PR[91,1] = PR[90,1] + -18.347;
   1:  PR[91,2] = PR[90,2] + 19.034;
   1:L PR[91] R[100]mm/sec CNT100;
   1:  PR[91,1] = PR[90,1] + -21.653;
   1:  PR[91,2] = PR[90,2] + 15.327;
   1:L PR[91] R[100]mm/sec CNT100;
   1:  PR[91,1] = PR[90,1] + -21.948;
   1:  PR[91,2] = PR[90,2] + 14.900;
   1:L PR[91] R[100]mm/sec CNT100;
   1:  PR[91,1] = PR[90,1] + -24.377;
   1:  PR[91,2] = PR[90,2] + 10.729;
   1:L PR[91] R[100]mm/sec CNT100;
   1:  PR[91,1] = PR[90,1] + -25.496;
   1:  PR[91,2] = PR[90,2] + 7.884;
   1:L PR[91] R[100]mm/sec CNT100;
   1:  PR[91,1] = PR[90,1] + -26.181;
   1:  PR[91,2] = PR[90,2] + 5.441;
   1:L PR[91] R[100]mm/sec CNT100;
   1:  PR[91,1] = PR[90,1] + -26.612;
   1:  PR[91,2] = PR[90,2] + 2.861;
   1:L PR[91] R[100]mm/sec CNT100;
   1:  PR[91,1] = PR[90,1] + -26.772;
   1:  PR[91,2] = PR[90,2] + -0.014;
   1:L PR[91] R[100]mm/sec CNT100;
   1:  PR[91,1] = PR[90,1] + -26.825;
   1:  PR[91,2] = PR[90,2] + -0.445;
   1:L PR[91] R[100]mm/sec CNT100;
   1:  PR[91,1] = PR[90,1] + -26.299;
   1:  PR[91,2] = PR[90,2] + -5.537;
   1:L PR[91] R[100]mm/sec CNT100;
   1:  PR[91,1] = PR[90,1] + -26.251;
   1:  PR[91,2] = PR[90,2] + -5.931;
   1:L PR[91] R[100]mm/sec CNT100;
   1:  PR[91,1] = PR[90,1] + -24.753;
   1:  PR[91,2] = PR[90,2] + -10.669;
   1:L PR[91] R[100]mm/sec CNT100;
   1:  PR[91,1] = PR[90,1] + -24.597;
   1:  PR[91,2] = PR[90,2] + -11.082;
   1:L PR[91] R[100]mm/sec CNT100;
   1:  PR[91,1] = PR[90,1] + -22.187;
   1:  PR[91,2] = PR[90,2] + -15.399;
   1:L PR[91] R[100]mm/sec CNT100;
   1:  PR[91,1] = PR[90,1] + -20.563;
   1:  PR[91,2] = PR[90,2] + -17.463;
   1:L PR[91] R[100]mm/sec CNT100;
   1:  PR[91,1] = PR[90,1] + -20.184;
   1:  PR[91,2] = PR[90,2] + -18.013;
   1:L PR[91] R[100]mm/sec CNT100;
   1:  PR[91,1] = PR[90,1] + -18.389;
   1:  PR[91,2] = PR[90,2] + -19.844;
   1:L PR[91] R[100]mm/sec CNT100;
   1:  PR[91,1] = PR[90,1] + -17.890;
   1:  PR[91,2] = PR[90,2] + -20.286;
   1:L PR[91] R[100]mm/sec CNT100;
   1:  PR[91,1] = PR[90,1] + -14.153;
   1:  PR[91,2] = PR[90,2] + -23.080;
   1:L PR[91] R[100]mm/sec CNT100;
   1:  PR[91,1] = PR[90,1] + -13.687;
   1:  PR[91,2] = PR[90,2] + -23.325;
   1:L PR[91] R[100]mm/sec CNT100;
   1:  PR[91,1] = PR[90,1] + -9.654;
   1:  PR[91,2] = PR[90,2] + -25.291;
   1:L PR[91] R[100]mm/sec CNT100;
   1:  PR[91,1] = PR[90,1] + -5.270;
   1:  PR[91,2] = PR[90,2] + -26.514;
   1:L PR[91] R[100]mm/sec CNT100;
   1:  PR[91,1] = PR[90,1] + -4.952;
   1:  PR[91,2] = PR[90,2] + -26.592;
   1:L PR[91] R[100]mm/sec CNT100;
   1:  PR[91,1] = PR[90,1] + -0.369;
   1:  PR[91,2] = PR[90,2] + -27.010;
   1:L PR[91] R[100]mm/sec CNT100;
   1:  PR[91,1] = PR[90,1] + -0.118;
   1:L PR[91] R[100]mm/sec CNT100;
   1:  PR[91,1] = PR[90,1] + 4.775;
   1:  PR[91,2] = PR[90,2] + -26.535;
   1:L PR[91] R[100]mm/sec CNT100;
   1:  PR[91,1] = PR[90,1] + 5.092;
   1:  PR[91,2] = PR[90,2] + -26.457;
   1:L PR[91] R[100]mm/sec CNT100;
   1:  PR[91,1] = PR[90,1] + 9.515;
   1:  PR[91,2] = PR[90,2] + -25.160;
   1:L PR[91] R[100]mm/sec CNT100;
   1:  PR[91,1] = PR[90,1] + 13.399;
   1:  PR[91,2] = PR[90,2] + -23.206;
   1:L PR[91] R[100]mm/sec CNT100;
   1:  PR[91,1] = PR[90,1] + 13.877;
   1:  PR[91,2] = PR[90,2] + -22.955;
   1:L PR[91] R[100]mm/sec CNT100;
   1:  PR[91,1] = PR[90,1] + 17.407;
   1:  PR[91,2] = PR[90,2] + -20.289;
   1:L PR[91] R[100]mm/sec CNT100;
   1:  PR[91,1] = PR[90,1] + 17.867;
   1:  PR[91,2] = PR[90,2] + -19.882;
   1:L PR[91] R[100]mm/sec CNT100;
   1:  PR[91,1] = PR[90,1] + 21.175;
   1:  PR[91,2] = PR[90,2] + -16.174;
   1:L PR[91] R[100]mm/sec CNT100;
   1:  PR[91,1] = PR[90,1] + 21.469;
   1:  PR[91,2] = PR[90,2] + -15.747;
   1:L PR[91] R[100]mm/sec CNT100;
   1:  PR[91,1] = PR[90,1] + 23.898;
   1:  PR[91,2] = PR[90,2] + -11.575;
   1:L PR[91] R[100]mm/sec CNT100;
   1:  PR[91,1] = PR[90,1] + 25.017;
   1:  PR[91,2] = PR[90,2] + -8.729;
   1:L PR[91] R[100]mm/sec CNT100;
   1:  PR[91,1] = PR[90,1] + 25.702;
   1:  PR[91,2] = PR[90,2] + -6.287;
   1:L PR[91] R[100]mm/sec CNT100;
   1:  PR[91,1] = PR[90,1] + 26.133;
   1:  PR[91,2] = PR[90,2] + -3.707;
   1:L PR[91] R[100]mm/sec CNT100;
   1:  PR[91,1] = PR[90,1] + 26.293;
   1:  PR[91,2] = PR[90,2] + -0.833;
   1:L PR[91] R[100]mm/sec CNT100;
   1:  PR[91,1] = PR[90,1] + 26.345;
   1:  PR[91,2] = PR[90,2] + -0.402;
   1:L PR[91] R[100]mm/sec CNT100;
   1:  PR[91,1] = PR[90,1] + 25.819;
   1:  PR[91,2] = PR[90,2] + 4.692;
   1:L PR[91] R[100]mm/sec CNT100;
   1:  PR[91,1] = PR[90,1] + 25.771;
   1:  PR[91,2] = PR[90,2] + 5.086;
   1:L PR[91] R[100]mm/sec CNT100;
   1:  PR[91,1] = PR[90,1] + 24.271;
   1:  PR[91,2] = PR[90,2] + 9.828;
   1:L PR[91] R[100]mm/sec CNT100;
   1:  PR[91,1] = PR[90,1] + 24.114;
   1:  PR[91,2] = PR[90,2] + 10.241;
   1:L PR[91] R[100]mm/sec CNT100;
   1:  PR[91,1] = PR[90,1] + 21.707;
   1:  PR[91,2] = PR[90,2] + 14.553;
   1:L PR[91] R[100]mm/sec CNT100;
   1:  PR[91,1] = PR[90,1] + 20.083;
   1:  PR[91,2] = PR[90,2] + 16.617;
   1:L PR[91] R[100]mm/sec CNT100;
   1:  PR[91,1] = PR[90,1] + 19.703;
   1:  PR[91,2] = PR[90,2] + 17.167;
   1:L PR[91] R[100]mm/sec CNT100;
   1:  PR[91,1] = PR[90,1] + 17.950;
   1:  PR[91,2] = PR[90,2] + 18.956;
   1:L PR[91] R[100]mm/sec CNT100;
   1:  PR[91,1] = PR[90,1] + 15.572;
   1:  PR[91,2] = PR[90,2] + 20.870;
   1:L PR[91] R[100]mm/sec CNT100;
   1:  PR[91,1] = PR[90,1] + 15.047;
   1:  PR[91,2] = PR[90,2] + 21.335;
   1:L PR[91] R[100]mm/sec CNT100;
   1:  PR[91,1] = PR[90,1] + 12.680;
   1:  PR[91,2] = PR[90,2] + 22.801;
   1:L PR[91] R[100]mm/sec CNT100;
   1:  PR[91,1] = PR[90,1] + 9.908;
   1:  PR[91,2] = PR[90,2] + 24.077;
   1:L PR[91] R[100]mm/sec CNT100;
   1:  PR[91,1] = PR[90,1] + 9.286;
   1:  PR[91,2] = PR[90,2] + 24.403;
   1:L PR[91] R[100]mm/sec CNT100;
   1:  PR[91,1] = PR[90,1] + 6.638;
   1:  PR[91,2] = PR[90,2] + 25.246;
   1:L PR[91] R[100]mm/sec CNT100;
   1:  PR[91,1] = PR[90,1] + 3.633;
   1:  PR[91,2] = PR[90,2] + 25.808;
   1:L PR[91] R[100]mm/sec CNT100;
   1:  PR[91,1] = PR[90,1] + 2.953;
   1:  PR[91,2] = PR[90,2] + 25.975;
   1:L PR[91] R[100]mm/sec CNT100;
   1:  PR[91,1] = PR[90,1] + 0.110;
   1:  PR[91,2] = PR[90,2] + 26.151;
   1:L PR[91] R[100]mm/sec CNT100;
   1:  PR[91] = PR[90];
   1:  PR[91,1] = PR[90,1] + -1.376;
   1:  PR[91,2] = PR[90,2] + 26.103;
   1:  PR[91,3] = PR[90,3] + 76.895;
   1:L PR[91] R[100]mm/sec CNT100;
   1:  PR[91,1] = PR[90,1] + -3.487;
   1:  PR[91,2] = PR[90,2] + 25.973;
   1:L PR[91] R[100]mm/sec CNT100;
   1:  PR[91,1] = PR[90,1] + -5.571;
   1:  PR[91,2] = PR[90,2] + 25.583;
   1:L PR[91] R[100]mm/sec CNT100;
   1:  PR[91,1] = PR[90,1] + -7.773;
   1:  PR[91,2] = PR[90,2] + 25.040;
   1:L PR[91] R[100]mm/sec CNT100;
   1:  PR[91,1] = PR[90,1] + -9.782;
   1:  PR[91,2] = PR[90,2] + 24.401;
   1:L PR[91] R[100]mm/sec CNT100;
   1:  PR[91,1] = PR[90,1] + -11.713;
   1:  PR[91,2] = PR[90,2] + 23.512;
   1:L PR[91] R[100]mm/sec CNT100;
   1:  PR[91,1] = PR[90,1] + -13.723;
   1:  PR[91,2] = PR[90,2] + 22.457;
   1:L PR[91] R[100]mm/sec CNT100;
   1:  PR[91,1] = PR[90,1] + -15.511;
   1:  PR[91,2] = PR[90,2] + 21.350;
   1:L PR[91] R[100]mm/sec CNT100;
   1:  PR[91,1] = PR[90,1] + -17.171;
   1:  PR[91,2] = PR[90,2] + 20.013;
   1:L PR[91] R[100]mm/sec CNT100;
   1:  PR[91,1] = PR[90,1] + -18.832;
   1:  PR[91,2] = PR[90,2] + 18.542;
   1:L PR[91] R[100]mm/sec CNT100;
   1:  PR[91,1] = PR[90,1] + -21.246;
   1:  PR[91,2] = PR[90,2] + 15.836;
   1:L PR[91] R[100]mm/sec CNT100;
   1:  PR[91,1] = PR[90,1] + -22.444;
   1:  PR[91,2] = PR[90,2] + 14.100;
   1:L PR[91] R[100]mm/sec CNT100;
   1:  PR[91,1] = PR[90,1] + -24.220;
   1:  PR[91,2] = PR[90,2] + 11.051;
   1:L PR[91] R[100]mm/sec CNT100;
   1:  PR[91,1] = PR[90,1] + -24.888;
   1:  PR[91,2] = PR[90,2] + 9.367;
   1:L PR[91] R[100]mm/sec CNT100;
   1:  PR[91,1] = PR[90,1] + -25.651;
   1:  PR[91,2] = PR[90,2] + 7.354;
   1:L PR[91] R[100]mm/sec CNT100;
   1:  PR[91,1] = PR[90,1] + -26.148;
   1:  PR[91,2] = PR[90,2] + 5.582;
   1:L PR[91] R[100]mm/sec CNT100;
   1:  PR[91,1] = PR[90,1] + -26.458;
   1:  PR[91,2] = PR[90,2] + 3.726;
   1:L PR[91] R[100]mm/sec CNT100;
   1:  PR[91,1] = PR[90,1] + -26.577;
   1:  PR[91,2] = PR[90,2] + 1.598;
   1:L PR[91] R[100]mm/sec CNT100;
   1:  PR[91,1] = PR[90,1] + -26.825;
   1:  PR[91,2] = PR[90,2] + -0.445;
   1:L PR[91] R[100]mm/sec CNT100;
   1:  PR[91,1] = PR[90,1] + -26.441;
   1:  PR[91,2] = PR[90,2] + -4.164;
   1:L PR[91] R[100]mm/sec CNT100;
   1:  PR[91,1] = PR[90,1] + -26.198;
   1:  PR[91,2] = PR[90,2] + -6.166;
   1:L PR[91] R[100]mm/sec CNT100;
   1:  PR[91,1] = PR[90,1] + -25.104;
   1:  PR[91,2] = PR[90,2] + -9.625;
   1:L PR[91] R[100]mm/sec CNT100;
   1:  PR[91,1] = PR[90,1] + -24.377;
   1:  PR[91,2] = PR[90,2] + -11.542;
   1:L PR[91] R[100]mm/sec CNT100;
   1:  PR[91,1] = PR[90,1] + -22.628;
   1:  PR[91,2] = PR[90,2] + -14.676;
   1:L PR[91] R[100]mm/sec CNT100;
   1:  PR[91,1] = PR[90,1] + -21.437;
   1:  PR[91,2] = PR[90,2] + -16.190;
   1:L PR[91] R[100]mm/sec CNT100;
   1:  PR[91,1] = PR[90,1] + -20.159;
   1:  PR[91,2] = PR[90,2] + -18.041;
   1:L PR[91] R[100]mm/sec CNT100;
   1:  PR[91,1] = PR[90,1] + -18.874;
   1:  PR[91,2] = PR[90,2] + -19.352;
   1:L PR[91] R[100]mm/sec CNT100;
   1:  PR[91,1] = PR[90,1] + -17.203;
   1:  PR[91,2] = PR[90,2] + -20.832;
   1:L PR[91] R[100]mm/sec CNT100;
   1:  PR[91,1] = PR[90,1] + -14.479;
   1:  PR[91,2] = PR[90,2] + -22.869;
   1:L PR[91] R[100]mm/sec CNT100;
   1:  PR[91,1] = PR[90,1] + -12.603;
   1:  PR[91,2] = PR[90,2] + -23.854;
   1:L PR[91] R[100]mm/sec CNT100;
   1:  PR[91,1] = PR[90,1] + -9.657;
   1:  PR[91,2] = PR[90,2] + -25.290;
   1:L PR[91] R[100]mm/sec CNT100;
   1:  PR[91,1] = PR[90,1] + -6.455;
   1:  PR[91,2] = PR[90,2] + -26.183;
   1:L PR[91] R[100]mm/sec CNT100;
   1:  PR[91,1] = PR[90,1] + -4.540;
   1:  PR[91,2] = PR[90,2] + -26.655;
   1:L PR[91] R[100]mm/sec CNT100;
   1:  PR[91,1] = PR[90,1] + -1.201;
   1:  PR[91,2] = PR[90,2] + -26.960;
   1:L PR[91] R[100]mm/sec CNT100;
   1:  PR[91,1] = PR[90,1] + 0.714;
   1:L PR[91] R[100]mm/sec CNT100;
   1:  PR[91,1] = PR[90,1] + 4.285;
   1:  PR[91,2] = PR[90,2] + -26.613;
   1:L PR[91] R[100]mm/sec CNT100;
   1:  PR[91,1] = PR[90,1] + 6.195;
   1:  PR[91,2] = PR[90,2] + -26.142;
   1:L PR[91] R[100]mm/sec CNT100;
   1:  PR[91,1] = PR[90,1] + 9.424;
   1:  PR[91,2] = PR[90,2] + -25.195;
   1:L PR[91] R[100]mm/sec CNT100;
   1:  PR[91,1] = PR[90,1] + 12.262;
   1:  PR[91,2] = PR[90,2] + -23.767;
   1:L PR[91] R[100]mm/sec CNT100;
   1:  PR[91,1] = PR[90,1] + 14.150;
   1:  PR[91,2] = PR[90,2] + -22.776;
   1:L PR[91] R[100]mm/sec CNT100;
   1:  PR[91,1] = PR[90,1] + 16.720;
   1:  PR[91,2] = PR[90,2] + -20.835;
   1:L PR[91] R[100]mm/sec CNT100;
   1:  PR[91,1] = PR[90,1] + 18.352;
   1:  PR[91,2] = PR[90,2] + -19.389;
   1:L PR[91] R[100]mm/sec CNT100;
   1:  PR[91,1] = PR[90,1] + 20.767;
   1:  PR[91,2] = PR[90,2] + -16.683;
   1:L PR[91] R[100]mm/sec CNT100;
   1:  PR[91,1] = PR[90,1] + 21.965;
   1:  PR[91,2] = PR[90,2] + -14.947;
   1:L PR[91] R[100]mm/sec CNT100;
   1:  PR[91,1] = PR[90,1] + 23.741;
   1:  PR[91,2] = PR[90,2] + -11.897;
   1:L PR[91] R[100]mm/sec CNT100;
   1:  PR[91,1] = PR[90,1] + 24.409;
   1:  PR[91,2] = PR[90,2] + -10.213;
   1:L PR[91] R[100]mm/sec CNT100;
   1:  PR[91,1] = PR[90,1] + 25.172;
   1:  PR[91,2] = PR[90,2] + -8.200;
   1:L PR[91] R[100]mm/sec CNT100;
   1:  PR[91,1] = PR[90,1] + 25.668;
   1:  PR[91,2] = PR[90,2] + -6.428;
   1:L PR[91] R[100]mm/sec CNT100;
   1:  PR[91,1] = PR[90,1] + 25.978;
   1:  PR[91,2] = PR[90,2] + -4.573;
   1:L PR[91] R[100]mm/sec CNT100;
   1:  PR[91,1] = PR[90,1] + 26.097;
   1:  PR[91,2] = PR[90,2] + -2.446;
   1:L PR[91] R[100]mm/sec CNT100;
   1:  PR[91,1] = PR[90,1] + 26.345;
   1:  PR[91,2] = PR[90,2] + -0.402;
   1:L PR[91] R[100]mm/sec CNT100;
   1:  PR[91,1] = PR[90,1] + 25.961;
   1:  PR[91,2] = PR[90,2] + 3.319;
   1:L PR[91] R[100]mm/sec CNT100;
   1:  PR[91,1] = PR[90,1] + 25.718;
   1:  PR[91,2] = PR[90,2] + 5.320;
   1:L PR[91] R[100]mm/sec CNT100;
   1:  PR[91,1] = PR[90,1] + 24.622;
   1:  PR[91,2] = PR[90,2] + 8.782;
   1:L PR[91] R[100]mm/sec CNT100;
   1:  PR[91,1] = PR[90,1] + 23.896;
   1:  PR[91,2] = PR[90,2] + 10.699;
   1:L PR[91] R[100]mm/sec CNT100;
   1:  PR[91,1] = PR[90,1] + 22.148;
   1:  PR[91,2] = PR[90,2] + 13.829;
   1:L PR[91] R[100]mm/sec CNT100;
   1:  PR[91,1] = PR[90,1] + 20.956;
   1:  PR[91,2] = PR[90,2] + 15.344;
   1:L PR[91] R[100]mm/sec CNT100;
   1:  PR[91,1] = PR[90,1] + 19.679;
   1:  PR[91,2] = PR[90,2] + 17.195;
   1:L PR[91] R[100]mm/sec CNT100;
   1:  PR[91,1] = PR[90,1] + 18.435;
   1:  PR[91,2] = PR[90,2] + 18.464;
   1:L PR[91] R[100]mm/sec CNT100;
   1:  PR[91,1] = PR[90,1] + 16.680;
   1:  PR[91,2] = PR[90,2] + 19.876;
   1:L PR[91] R[100]mm/sec CNT100;
   1:  PR[91,1] = PR[90,1] + 14.983;
   1:  PR[91,2] = PR[90,2] + 21.380;
   1:L PR[91] R[100]mm/sec CNT100;
   1:  PR[91,1] = PR[90,1] + 13.297;
   1:  PR[91,2] = PR[90,2] + 22.424;
   1:L PR[91] R[100]mm/sec CNT100;
   1:  PR[91,1] = PR[90,1] + 11.252;
   1:  PR[91,2] = PR[90,2] + 23.365;
   1:L PR[91] R[100]mm/sec CNT100;
   1:  PR[91,1] = PR[90,1] + 9.242;
   1:  PR[91,2] = PR[90,2] + 24.420;
   1:L PR[91] R[100]mm/sec CNT100;
   1:  PR[91,1] = PR[90,1] + 7.357;
   1:  PR[91,2] = PR[90,2] + 25.020;
   1:L PR[91] R[100]mm/sec CNT100;
   1:  PR[91,1] = PR[90,1] + 5.139;
   1:  PR[91,2] = PR[90,2] + 25.434;
   1:L PR[91] R[100]mm/sec CNT100;
   1:  PR[91,1] = PR[90,1] + 2.937;
   1:  PR[91,2] = PR[90,2] + 25.977;
   1:L PR[91] R[100]mm/sec CNT100;
   1:  PR[91,1] = PR[90,1] + 0.894;
   1:  PR[91,2] = PR[90,2] + 26.103;
   1:L PR[91] R[100]mm/sec CNT100;
   1:  PR[91] = PR[90];
   1:  PR[91,1] = PR[90,1] + -2.159;
   1:  PR[91,2] = PR[90,2] + 26.056;
   1:  PR[91,3] = PR[90,3] + 78.195;
   1:L PR[91] R[100]mm/sec CNT100;
   1:  PR[91,1] = PR[90,1] + -3.471;
   1:  PR[91,2] = PR[90,2] + 25.975;
   1:L PR[91] R[100]mm/sec CNT100;
   1:  PR[91,1] = PR[90,1] + -4.768;
   1:  PR[91,2] = PR[90,2] + 25.732;
   1:L PR[91] R[100]mm/sec CNT100;
   1:  PR[91,1] = PR[90,1] + -8.491;
   1:  PR[91,2] = PR[90,2] + 24.814;
   1:L PR[91] R[100]mm/sec CNT100;
   1:  PR[91,1] = PR[90,1] + -9.738;
   1:  PR[91,2] = PR[90,2] + 24.418;
   1:L PR[91] R[100]mm/sec CNT100;
   1:  PR[91,1] = PR[90,1] + -10.942;
   1:  PR[91,2] = PR[90,2] + 23.863;
   1:L PR[91] R[100]mm/sec CNT100;
   1:  PR[91,1] = PR[90,1] + -14.340;
   1:  PR[91,2] = PR[90,2] + 22.080;
   1:L PR[91] R[100]mm/sec CNT100;
   1:  PR[91,1] = PR[90,1] + -15.447;
   1:  PR[91,2] = PR[90,2] + 21.394;
   1:L PR[91] R[100]mm/sec CNT100;
   1:  PR[91,1] = PR[90,1] + -16.484;
   1:  PR[91,2] = PR[90,2] + 20.560;
   1:L PR[91] R[100]mm/sec CNT100;
   1:  PR[91,1] = PR[90,1] + -19.317;
   1:  PR[91,2] = PR[90,2] + 18.050;
   1:L PR[91] R[100]mm/sec CNT100;
   1:  PR[91,1] = PR[90,1] + -20.838;
   1:  PR[91,2] = PR[90,2] + 16.345;
   1:L PR[91] R[100]mm/sec CNT100;
   1:  PR[91,1] = PR[90,1] + -22.940;
   1:  PR[91,2] = PR[90,2] + 13.300;
   1:L PR[91] R[100]mm/sec CNT100;
   1:  PR[91,1] = PR[90,1] + -24.060;
   1:  PR[91,2] = PR[90,2] + 11.376;
   1:L PR[91] R[100]mm/sec CNT100;
   1:  PR[91,1] = PR[90,1] + -24.475;
   1:  PR[91,2] = PR[90,2] + 10.332;
   1:L PR[91] R[100]mm/sec CNT100;
   1:  PR[91,1] = PR[90,1] + -25.810;
   1:  PR[91,2] = PR[90,2] + 6.810;
   1:L PR[91] R[100]mm/sec CNT100;
   1:  PR[91,1] = PR[90,1] + -26.115;
   1:  PR[91,2] = PR[90,2] + 5.723;
   1:L PR[91] R[100]mm/sec CNT100;
   1:  PR[91,1] = PR[90,1] + -26.304;
   1:  PR[91,2] = PR[90,2] + 4.591;
   1:L PR[91] R[100]mm/sec CNT100;
   1:  PR[91,1] = PR[90,1] + -26.381;
   1:  PR[91,2] = PR[90,2] + 3.211;
   1:L PR[91] R[100]mm/sec CNT100;
   1:  PR[91,1] = PR[90,1] + -26.825;
   1:  PR[91,2] = PR[90,2] + -0.445;
   1:L PR[91] R[100]mm/sec CNT100;
   1:  PR[91,1] = PR[90,1] + -26.583;
   1:  PR[91,2] = PR[90,2] + -2.791;
   1:L PR[91] R[100]mm/sec CNT100;
   1:  PR[91,1] = PR[90,1] + -26.144;
   1:  PR[91,2] = PR[90,2] + -6.402;
   1:L PR[91] R[100]mm/sec CNT100;
   1:  PR[91,1] = PR[90,1] + -25.455;
   1:  PR[91,2] = PR[90,2] + -8.580;
   1:L PR[91] R[100]mm/sec CNT100;
   1:  PR[91,1] = PR[90,1] + -24.158;
   1:  PR[91,2] = PR[90,2] + -12.001;
   1:L PR[91] R[100]mm/sec CNT100;
   1:  PR[91,1] = PR[90,1] + -23.069;
   1:  PR[91,2] = PR[90,2] + -13.953;
   1:L PR[91] R[100]mm/sec CNT100;
   1:  PR[91,1] = PR[90,1] + -22.310;
   1:  PR[91,2] = PR[90,2] + -14.917;
   1:L PR[91] R[100]mm/sec CNT100;
   1:  PR[91,1] = PR[90,1] + -20.135;
   1:  PR[91,2] = PR[90,2] + -18.069;
   1:L PR[91] R[100]mm/sec CNT100;
   1:  PR[91,1] = PR[90,1] + -19.360;
   1:  PR[91,2] = PR[90,2] + -18.859;
   1:L PR[91] R[100]mm/sec CNT100;
   1:  PR[91,1] = PR[90,1] + -16.516;
   1:  PR[91,2] = PR[90,2] + -21.378;
   1:L PR[91] R[100]mm/sec CNT100;
   1:  PR[91,1] = PR[90,1] + -14.805;
   1:  PR[91,2] = PR[90,2] + -22.658;
   1:L PR[91] R[100]mm/sec CNT100;
   1:  PR[91,1] = PR[90,1] + -11.519;
   1:  PR[91,2] = PR[90,2] + -24.383;
   1:L PR[91] R[100]mm/sec CNT100;
   1:  PR[91,1] = PR[90,1] + -9.661;
   1:  PR[91,2] = PR[90,2] + -25.289;
   1:L PR[91] R[100]mm/sec CNT100;
   1:  PR[91,1] = PR[90,1] + -7.639;
   1:  PR[91,2] = PR[90,2] + -25.852;
   1:L PR[91] R[100]mm/sec CNT100;
   1:  PR[91,1] = PR[90,1] + -4.129;
   1:  PR[91,2] = PR[90,2] + -26.718;
   1:L PR[91] R[100]mm/sec CNT100;
   1:  PR[91,1] = PR[90,1] + -2.032;
   1:  PR[91,2] = PR[90,2] + -26.909;
   1:L PR[91] R[100]mm/sec CNT100;
   1:  PR[91,1] = PR[90,1] + 1.545;
   1:L PR[91] R[100]mm/sec CNT100;
   1:  PR[91,1] = PR[90,1] + 3.794;
   1:  PR[91,2] = PR[90,2] + -26.690;
   1:L PR[91] R[100]mm/sec CNT100;
   1:  PR[91,1] = PR[90,1] + 7.299;
   1:  PR[91,2] = PR[90,2] + -25.827;
   1:L PR[91] R[100]mm/sec CNT100;
   1:  PR[91,1] = PR[90,1] + 9.333;
   1:  PR[91,2] = PR[90,2] + -25.230;
   1:L PR[91] R[100]mm/sec CNT100;
   1:  PR[91,1] = PR[90,1] + 11.126;
   1:  PR[91,2] = PR[90,2] + -24.328;
   1:L PR[91] R[100]mm/sec CNT100;
   1:  PR[91,1] = PR[90,1] + 14.423;
   1:  PR[91,2] = PR[90,2] + -22.598;
   1:L PR[91] R[100]mm/sec CNT100;
   1:  PR[91,1] = PR[90,1] + 16.033;
   1:  PR[91,2] = PR[90,2] + -21.382;
   1:L PR[91] R[100]mm/sec CNT100;
   1:  PR[91,1] = PR[90,1] + 18.838;
   1:  PR[91,2] = PR[90,2] + -18.897;
   1:L PR[91] R[100]mm/sec CNT100;
   1:  PR[91,1] = PR[90,1] + 20.359;
   1:  PR[91,2] = PR[90,2] + -17.192;
   1:L PR[91] R[100]mm/sec CNT100;
   1:  PR[91,1] = PR[90,1] + 22.460;
   1:  PR[91,2] = PR[90,2] + -14.147;
   1:L PR[91] R[100]mm/sec CNT100;
   1:  PR[91,1] = PR[90,1] + 23.581;
   1:  PR[91,2] = PR[90,2] + -12.223;
   1:L PR[91] R[100]mm/sec CNT100;
   1:  PR[91,1] = PR[90,1] + 23.995;
   1:  PR[91,2] = PR[90,2] + -11.179;
   1:L PR[91] R[100]mm/sec CNT100;
   1:  PR[91,1] = PR[90,1] + 25.331;
   1:  PR[91,2] = PR[90,2] + -7.657;
   1:L PR[91] R[100]mm/sec CNT100;
   1:  PR[91,1] = PR[90,1] + 25.635;
   1:  PR[91,2] = PR[90,2] + -6.569;
   1:L PR[91] R[100]mm/sec CNT100;
   1:  PR[91,1] = PR[90,1] + 25.824;
   1:  PR[91,2] = PR[90,2] + -5.438;
   1:L PR[91] R[100]mm/sec CNT100;
   1:  PR[91,1] = PR[90,1] + 25.901;
   1:  PR[91,2] = PR[90,2] + -4.058;
   1:L PR[91] R[100]mm/sec CNT100;
   1:  PR[91,1] = PR[90,1] + 26.345;
   1:  PR[91,2] = PR[90,2] + -0.402;
   1:L PR[91] R[100]mm/sec CNT100;
   1:  PR[91,1] = PR[90,1] + 26.103;
   1:  PR[91,2] = PR[90,2] + 1.945;
   1:L PR[91] R[100]mm/sec CNT100;
   1:  PR[91,1] = PR[90,1] + 25.664;
   1:  PR[91,2] = PR[90,2] + 5.555;
   1:L PR[91] R[100]mm/sec CNT100;
   1:  PR[91,1] = PR[90,1] + 24.974;
   1:  PR[91,2] = PR[90,2] + 7.736;
   1:L PR[91] R[100]mm/sec CNT100;
   1:  PR[91,1] = PR[90,1] + 23.677;
   1:  PR[91,2] = PR[90,2] + 11.157;
   1:L PR[91] R[100]mm/sec CNT100;
   1:  PR[91,1] = PR[90,1] + 22.589;
   1:  PR[91,2] = PR[90,2] + 13.106;
   1:L PR[91] R[100]mm/sec CNT100;
   1:  PR[91,1] = PR[90,1] + 21.830;
   1:  PR[91,2] = PR[90,2] + 14.071;
   1:L PR[91] R[100]mm/sec CNT100;
   1:  PR[91,1] = PR[90,1] + 19.654;
   1:  PR[91,2] = PR[90,2] + 17.222;
   1:L PR[91] R[100]mm/sec CNT100;
   1:  PR[91,1] = PR[90,1] + 18.920;
   1:  PR[91,2] = PR[90,2] + 17.971;
   1:L PR[91] R[100]mm/sec CNT100;
   1:  PR[91,1] = PR[90,1] + 17.789;
   1:  PR[91,2] = PR[90,2] + 18.882;
   1:L PR[91] R[100]mm/sec CNT100;
   1:  PR[91,1] = PR[90,1] + 14.919;
   1:  PR[91,2] = PR[90,2] + 21.424;
   1:L PR[91] R[100]mm/sec CNT100;
   1:  PR[91,1] = PR[90,1] + 13.914;
   1:  PR[91,2] = PR[90,2] + 22.047;
   1:L PR[91] R[100]mm/sec CNT100;
   1:  PR[91,1] = PR[90,1] + 12.596;
   1:  PR[91,2] = PR[90,2] + 22.654;
   1:L PR[91] R[100]mm/sec CNT100;
   1:  PR[91,1] = PR[90,1] + 9.198;
   1:  PR[91,2] = PR[90,2] + 24.437;
   1:L PR[91] R[100]mm/sec CNT100;
   1:  PR[91,1] = PR[90,1] + 8.076;
   1:  PR[91,2] = PR[90,2] + 24.794;
   1:L PR[91] R[100]mm/sec CNT100;
   1:  PR[91,1] = PR[90,1] + 6.644;
   1:  PR[91,2] = PR[90,2] + 25.061;
   1:L PR[91] R[100]mm/sec CNT100;
   1:  PR[91,1] = PR[90,1] + 2.922;
   1:  PR[91,2] = PR[90,2] + 25.979;
   1:L PR[91] R[100]mm/sec CNT100;
   1:  PR[91,1] = PR[90,1] + 1.679;
   1:  PR[91,2] = PR[90,2] + 26.056;
   1:L PR[91] R[100]mm/sec CNT100;
   1:  PR[91] = PR[90];
   1:  PR[91,1] = PR[90,1] + -2.943;
   1:  PR[91,2] = PR[90,2] + 26.008;
   1:  PR[91,3] = PR[90,3] + 79.495;
   1:L PR[91] R[100]mm/sec CNT100;
   1:  PR[91,1] = PR[90,1] + -3.456;
   1:  PR[91,2] = PR[90,2] + 25.976;
   1:L PR[91] R[100]mm/sec CNT100;
   1:  PR[91,1] = PR[90,1] + -3.966;
   1:  PR[91,2] = PR[90,2] + 25.881;
   1:L PR[91] R[100]mm/sec CNT100;
   1:  PR[91,1] = PR[90,1] + -9.210;
   1:  PR[91,2] = PR[90,2] + 24.588;
   1:L PR[91] R[100]mm/sec CNT100;
   1:  PR[91,1] = PR[90,1] + -9.694;
   1:  PR[91,2] = PR[90,2] + 24.434;
   1:L PR[91] R[100]mm/sec CNT100;
   1:  PR[91,1] = PR[90,1] + -10.171;
   1:  PR[91,2] = PR[90,2] + 24.215;
   1:L PR[91] R[100]mm/sec CNT100;
   1:  PR[91,1] = PR[90,1] + -14.957;
   1:  PR[91,2] = PR[90,2] + 21.703;
   1:L PR[91] R[100]mm/sec CNT100;
   1:  PR[91,1] = PR[90,1] + -15.384;
   1:  PR[91,2] = PR[90,2] + 21.439;
   1:L PR[91] R[100]mm/sec CNT100;
   1:  PR[91,1] = PR[90,1] + -15.797;
   1:  PR[91,2] = PR[90,2] + 21.106;
   1:L PR[91] R[100]mm/sec CNT100;
   1:  PR[91,1] = PR[90,1] + -19.803;
   1:  PR[91,2] = PR[90,2] + 17.557;
   1:L PR[91] R[100]mm/sec CNT100;
   1:  PR[91,1] = PR[90,1] + -20.430;
   1:  PR[91,2] = PR[90,2] + 16.854;
   1:L PR[91] R[100]mm/sec CNT100;
   1:  PR[91,1] = PR[90,1] + -23.435;
   1:  PR[91,2] = PR[90,2] + 12.500;
   1:L PR[91] R[100]mm/sec CNT100;
   1:  PR[91,1] = PR[90,1] + -23.892;
   1:  PR[91,2] = PR[90,2] + 11.716;
   1:L PR[91] R[100]mm/sec CNT100;
   1:  PR[91,1] = PR[90,1] + -25.969;
   1:  PR[91,2] = PR[90,2] + 6.264;
   1:L PR[91] R[100]mm/sec CNT100;
   1:  PR[91,1] = PR[90,1] + -26.081;
   1:  PR[91,2] = PR[90,2] + 5.864;
   1:L PR[91] R[100]mm/sec CNT100;
   1:  PR[91,1] = PR[90,1] + -26.150;
   1:  PR[91,2] = PR[90,2] + 5.456;
   1:L PR[91] R[100]mm/sec CNT100;
   1:  PR[91,1] = PR[90,1] + -26.185;
   1:  PR[91,2] = PR[90,2] + 4.823;
   1:L PR[91] R[100]mm/sec CNT100;
   1:  PR[91,1] = PR[90,1] + -26.825;
   1:  PR[91,2] = PR[90,2] + -0.445;
   1:L PR[91] R[100]mm/sec CNT100;
   1:  PR[91,1] = PR[90,1] + -26.724;
   1:  PR[91,2] = PR[90,2] + -1.418;
   1:L PR[91] R[100]mm/sec CNT100;
   1:  PR[91,1] = PR[90,1] + -26.090;
   1:  PR[91,2] = PR[90,2] + -6.637;
   1:L PR[91] R[100]mm/sec CNT100;
   1:  PR[91,1] = PR[90,1] + -25.806;
   1:  PR[91,2] = PR[90,2] + -7.536;
   1:L PR[91] R[100]mm/sec CNT100;
   1:  PR[91,1] = PR[90,1] + -23.939;
   1:  PR[91,2] = PR[90,2] + -12.461;
   1:L PR[91] R[100]mm/sec CNT100;
   1:  PR[91,1] = PR[90,1] + -23.510;
   1:  PR[91,2] = PR[90,2] + -13.229;
   1:L PR[91] R[100]mm/sec CNT100;
   1:  PR[91,1] = PR[90,1] + -23.183;
   1:  PR[91,2] = PR[90,2] + -13.645;
   1:L PR[91] R[100]mm/sec CNT100;
   1:  PR[91,1] = PR[90,1] + -20.110;
   1:  PR[91,2] = PR[90,2] + -18.096;
   1:L PR[91] R[100]mm/sec CNT100;
   1:  PR[91,1] = PR[90,1] + -19.845;
   1:  PR[91,2] = PR[90,2] + -18.367;
   1:L PR[91] R[100]mm/sec CNT100;
   1:  PR[91,1] = PR[90,1] + -15.829;
   1:  PR[91,2] = PR[90,2] + -21.925;
   1:L PR[91] R[100]mm/sec CNT100;
   1:  PR[91,1] = PR[90,1] + -15.131;
   1:  PR[91,2] = PR[90,2] + -22.447;
   1:L PR[91] R[100]mm/sec CNT100;
   1:  PR[91,1] = PR[90,1] + -10.435;
   1:  PR[91,2] = PR[90,2] + -24.911;
   1:L PR[91] R[100]mm/sec CNT100;
   1:  PR[91,1] = PR[90,1] + -9.664;
   1:  PR[91,2] = PR[90,2] + -25.287;
   1:L PR[91] R[100]mm/sec CNT100;
   1:  PR[91,1] = PR[90,1] + -8.824;
   1:  PR[91,2] = PR[90,2] + -25.522;
   1:L PR[91] R[100]mm/sec CNT100;
   1:  PR[91,1] = PR[90,1] + -3.718;
   1:  PR[91,2] = PR[90,2] + -26.780;
   1:L PR[91] R[100]mm/sec CNT100;
   1:  PR[91,1] = PR[90,1] + -2.856;
   1:  PR[91,2] = PR[90,2] + -26.858;
   1:L PR[91] R[100]mm/sec CNT100;
   1:  PR[91,1] = PR[90,1] + 2.377;
   1:L PR[91] R[100]mm/sec CNT100;
   1:  PR[91,1] = PR[90,1] + 3.303;
   1:  PR[91,2] = PR[90,2] + -26.768;
   1:L PR[91] R[100]mm/sec CNT100;
   1:  PR[91,1] = PR[90,1] + 8.402;
   1:  PR[91,2] = PR[90,2] + -25.511;
   1:L PR[91] R[100]mm/sec CNT100;
   1:  PR[91,1] = PR[90,1] + 9.242;
   1:  PR[91,2] = PR[90,2] + -25.265;
   1:L PR[91] R[100]mm/sec CNT100;
   1:  PR[91,1] = PR[90,1] + 9.990;
   1:  PR[91,2] = PR[90,2] + -24.889;
   1:L PR[91] R[100]mm/sec CNT100;
   1:  PR[91,1] = PR[90,1] + 14.695;
   1:  PR[91,2] = PR[90,2] + -22.419;
   1:L PR[91] R[100]mm/sec CNT100;
   1:  PR[91,1] = PR[90,1] + 15.346;
   1:  PR[91,2] = PR[90,2] + -21.928;
   1:L PR[91] R[100]mm/sec CNT100;
   1:  PR[91,1] = PR[90,1] + 19.323;
   1:  PR[91,2] = PR[90,2] + -18.404;
   1:L PR[91] R[100]mm/sec CNT100;
   1:  PR[91,1] = PR[90,1] + 19.951;
   1:  PR[91,2] = PR[90,2] + -17.701;
   1:L PR[91] R[100]mm/sec CNT100;
   1:  PR[91,1] = PR[90,1] + 22.956;
   1:  PR[91,2] = PR[90,2] + -13.347;
   1:L PR[91] R[100]mm/sec CNT100;
   1:  PR[91,1] = PR[90,1] + 23.413;
   1:  PR[91,2] = PR[90,2] + -12.562;
   1:L PR[91] R[100]mm/sec CNT100;
   1:  PR[91,1] = PR[90,1] + 25.490;
   1:  PR[91,2] = PR[90,2] + -7.111;
   1:L PR[91] R[100]mm/sec CNT100;
   1:  PR[91,1] = PR[90,1] + 25.602;
   1:  PR[91,2] = PR[90,2] + -6.711;
   1:L PR[91] R[100]mm/sec CNT100;
   1:  PR[91,1] = PR[90,1] + 25.670;
   1:  PR[91,2] = PR[90,2] + -6.303;
   1:L PR[91] R[100]mm/sec CNT100;
   1:  PR[91,1] = PR[90,1] + 25.705;
   1:  PR[91,2] = PR[90,2] + -5.670;
   1:L PR[91] R[100]mm/sec CNT100;
   1:  PR[91,1] = PR[90,1] + 26.345;
   1:  PR[91,2] = PR[90,2] + -0.402;
   1:L PR[91] R[100]mm/sec CNT100;
   1:  PR[91,1] = PR[90,1] + 26.245;
   1:  PR[91,2] = PR[90,2] + 0.571;
   1:L PR[91] R[100]mm/sec CNT100;
   1:  PR[91,1] = PR[90,1] + 25.611;
   1:  PR[91,2] = PR[90,2] + 5.790;
   1:L PR[91] R[100]mm/sec CNT100;
   1:  PR[91,1] = PR[90,1] + 25.326;
   1:  PR[91,2] = PR[90,2] + 6.690;
   1:L PR[91] R[100]mm/sec CNT100;
   1:  PR[91,1] = PR[90,1] + 23.458;
   1:  PR[91,2] = PR[90,2] + 11.615;
   1:L PR[91] R[100]mm/sec CNT100;
   1:  PR[91,1] = PR[90,1] + 23.030;
   1:  PR[91,2] = PR[90,2] + 12.382;
   1:L PR[91] R[100]mm/sec CNT100;
   1:  PR[91,1] = PR[90,1] + 22.703;
   1:  PR[91,2] = PR[90,2] + 12.798;
   1:L PR[91] R[100]mm/sec CNT100;
   1:  PR[91,1] = PR[90,1] + 19.630;
   1:  PR[91,2] = PR[90,2] + 17.249;
   1:L PR[91] R[100]mm/sec CNT100;
   1:  PR[91,1] = PR[90,1] + 19.405;
   1:  PR[91,2] = PR[90,2] + 17.479;
   1:L PR[91] R[100]mm/sec CNT100;
   1:  PR[91,1] = PR[90,1] + 18.898;
   1:  PR[91,2] = PR[90,2] + 17.887;
   1:L PR[91] R[100]mm/sec CNT100;
   1:  PR[91,1] = PR[90,1] + 14.856;
   1:  PR[91,2] = PR[90,2] + 21.469;
   1:L PR[91] R[100]mm/sec CNT100;
   1:  PR[91,1] = PR[90,1] + 14.530;
   1:  PR[91,2] = PR[90,2] + 21.670;
   1:L PR[91] R[100]mm/sec CNT100;
   1:  PR[91,1] = PR[90,1] + 13.940;
   1:  PR[91,2] = PR[90,2] + 21.942;
   1:L PR[91] R[100]mm/sec CNT100;
   1:  PR[91,1] = PR[90,1] + 9.154;
   1:  PR[91,2] = PR[90,2] + 24.454;
   1:L PR[91] R[100]mm/sec CNT100;
   1:  PR[91,1] = PR[90,1] + 8.795;
   1:  PR[91,2] = PR[90,2] + 24.568;
   1:L PR[91] R[100]mm/sec CNT100;
   1:  PR[91,1] = PR[90,1] + 8.150;
   1:  PR[91,2] = PR[90,2] + 24.688;
   1:L PR[91] R[100]mm/sec CNT100;
   1:  PR[91,1] = PR[90,1] + 2.907;
   1:  PR[91,2] = PR[90,2] + 25.981;
   1:L PR[91] R[100]mm/sec CNT100;
   1:  PR[91,1] = PR[90,1] + 2.463;
   1:  PR[91,2] = PR[90,2] + 26.008;
   1:L PR[91] R[100]mm/sec CNT100;
   1:  PR[91,1] = PR[90,1] + -2.943;
   1:L PR[91] R[100]mm/sec CNT100;
   1:  PR[91,1] = PR[90,1] + -3.456;
   1:  PR[91,2] = PR[90,2] + 25.976;
   1:L PR[91] R[100]mm/sec CNT100;
   1:  PR[91,1] = PR[90,1] + -3.966;
   1:  PR[91,2] = PR[90,2] + 25.881;
   1:L PR[91] R[100]mm/sec CNT100;
   1:  PR[91,1] = PR[90,1] + -9.210;
   1:  PR[91,2] = PR[90,2] + 24.588;
   1:L PR[91] R[100]mm/sec CNT100;
   1:  PR[91,1] = PR[90,1] + -9.694;
   1:  PR[91,2] = PR[90,2] + 24.434;
   1:L PR[91] R[100]mm/sec CNT100;
   1:  PR[91,1] = PR[90,1] + -10.171;
   1:  PR[91,2] = PR[90,2] + 24.215;
   1:L PR[91] R[100]mm/sec CNT100;
   1:  PR[91,1] = PR[90,1] + -14.957;
   1:  PR[91,2] = PR[90,2] + 21.703;
   1:L PR[91] R[100]mm/sec CNT100;
   1:  PR[91,1] = PR[90,1] + -15.384;
   1:  PR[91,2] = PR[90,2] + 21.439;
   1:L PR[91] R[100]mm/sec CNT100;
   1:  PR[91,1] = PR[90,1] + -15.797;
   1:  PR[91,2] = PR[90,2] + 21.106;
   1:L PR[91] R[100]mm/sec CNT100;
   1:  PR[91,1] = PR[90,1] + -19.803;
   1:  PR[91,2] = PR[90,2] + 17.557;
   1:L PR[91] R[100]mm/sec CNT100;
   1:  PR[91,1] = PR[90,1] + -20.430;
   1:  PR[91,2] = PR[90,2] + 16.854;
   1:L PR[91] R[100]mm/sec CNT100;
   1:  PR[91,1] = PR[90,1] + -23.435;
   1:  PR[91,2] = PR[90,2] + 12.500;
   1:L PR[91] R[100]mm/sec CNT100;
   1:  PR[91,1] = PR[90,1] + -23.892;
   1:  PR[91,2] = PR[90,2] + 11.716;
   1:L PR[91] R[100]mm/sec CNT100;
   1:  PR[91,1] = PR[90,1] + -25.969;
   1:  PR[91,2] = PR[90,2] + 6.264;
   1:L PR[91] R[100]mm/sec CNT100;
   1:  PR[91,1] = PR[90,1] + -26.081;
   1:  PR[91,2] = PR[90,2] + 5.864;
   1:L PR[91] R[100]mm/sec CNT100;
   1:  PR[91,1] = PR[90,1] + -26.150;
   1:  PR[91,2] = PR[90,2] + 5.456;
   1:L PR[91] R[100]mm/sec CNT100;
   1:  PR[91,1] = PR[90,1] + -26.185;
   1:  PR[91,2] = PR[90,2] + 4.823;
   1:L PR[91] R[100]mm/sec CNT100;
   1:  PR[91,1] = PR[90,1] + -26.825;
   1:  PR[91,2] = PR[90,2] + -0.445;
   1:L PR[91] R[100]mm/sec CNT100;
   1:  PR[91,1] = PR[90,1] + -26.724;
   1:  PR[91,2] = PR[90,2] + -1.418;
   1:L PR[91] R[100]mm/sec CNT100;
   1:  PR[91,1] = PR[90,1] + -26.090;
   1:  PR[91,2] = PR[90,2] + -6.637;
   1:L PR[91] R[100]mm/sec CNT100;
   1:  PR[91,1] = PR[90,1] + -25.806;
   1:  PR[91,2] = PR[90,2] + -7.536;
   1:L PR[91] R[100]mm/sec CNT100;
   1:  PR[91,1] = PR[90,1] + -23.939;
   1:  PR[91,2] = PR[90,2] + -12.461;
   1:L PR[91] R[100]mm/sec CNT100;
   1:  PR[91,1] = PR[90,1] + -23.510;
   1:  PR[91,2] = PR[90,2] + -13.229;
   1:L PR[91] R[100]mm/sec CNT100;
   1:  PR[91,1] = PR[90,1] + -23.183;
   1:  PR[91,2] = PR[90,2] + -13.645;
   1:L PR[91] R[100]mm/sec CNT100;
   1:  PR[91,1] = PR[90,1] + -20.110;
   1:  PR[91,2] = PR[90,2] + -18.096;
   1:L PR[91] R[100]mm/sec CNT100;
   1:  PR[91,1] = PR[90,1] + -19.845;
   1:  PR[91,2] = PR[90,2] + -18.367;
   1:L PR[91] R[100]mm/sec CNT100;
   1:  PR[91,1] = PR[90,1] + -15.829;
   1:  PR[91,2] = PR[90,2] + -21.925;
   1:L PR[91] R[100]mm/sec CNT100;
   1:  PR[91,1] = PR[90,1] + -15.131;
   1:  PR[91,2] = PR[90,2] + -22.447;
   1:L PR[91] R[100]mm/sec CNT100;
   1:  PR[91,1] = PR[90,1] + -10.435;
   1:  PR[91,2] = PR[90,2] + -24.911;
   1:L PR[91] R[100]mm/sec CNT100;
   1:  PR[91,1] = PR[90,1] + -9.664;
   1:  PR[91,2] = PR[90,2] + -25.287;
   1:L PR[91] R[100]mm/sec CNT100;
   1:  PR[91,1] = PR[90,1] + -8.824;
   1:  PR[91,2] = PR[90,2] + -25.522;
   1:L PR[91] R[100]mm/sec CNT100;
   1:  PR[91,1] = PR[90,1] + -3.718;
   1:  PR[91,2] = PR[90,2] + -26.780;
   1:L PR[91] R[100]mm/sec CNT100;
   1:  PR[91,1] = PR[90,1] + -2.856;
   1:  PR[91,2] = PR[90,2] + -26.858;
   1:L PR[91] R[100]mm/sec CNT100;
   1:  PR[91,1] = PR[90,1] + 2.377;
   1:L PR[91] R[100]mm/sec CNT100;
   1:  PR[91,1] = PR[90,1] + 3.303;
   1:  PR[91,2] = PR[90,2] + -26.768;
   1:L PR[91] R[100]mm/sec CNT100;
   1:  PR[91,1] = PR[90,1] + 8.402;
   1:  PR[91,2] = PR[90,2] + -25.511;
   1:L PR[91] R[100]mm/sec CNT100;
   1:  PR[91,1] = PR[90,1] + 9.242;
   1:  PR[91,2] = PR[90,2] + -25.265;
   1:L PR[91] R[100]mm/sec CNT100;
   1:  PR[91,1] = PR[90,1] + 9.990;
   1:  PR[91,2] = PR[90,2] + -24.889;
   1:L PR[91] R[100]mm/sec CNT100;
   1:  PR[91,1] = PR[90,1] + 14.695;
   1:  PR[91,2] = PR[90,2] + -22.419;
   1:L PR[91] R[100]mm/sec CNT100;
   1:  PR[91,1] = PR[90,1] + 15.346;
   1:  PR[91,2] = PR[90,2] + -21.928;
   1:L PR[91] R[100]mm/sec CNT100;
   1:  PR[91,1] = PR[90,1] + 19.323;
   1:  PR[91,2] = PR[90,2] + -18.404;
   1:L PR[91] R[100]mm/sec CNT100;
   1:  PR[91,1] = PR[90,1] + 19.951;
   1:  PR[91,2] = PR[90,2] + -17.701;
   1:L PR[91] R[100]mm/sec CNT100;
   1:  PR[91,1] = PR[90,1] + 22.956;
   1:  PR[91,2] = PR[90,2] + -13.347;
   1:L PR[91] R[100]mm/sec CNT100;
   1:  PR[91,1] = PR[90,1] + 23.413;
   1:  PR[91,2] = PR[90,2] + -12.562;
   1:L PR[91] R[100]mm/sec CNT100;
   1:  PR[91,1] = PR[90,1] + 25.490;
   1:  PR[91,2] = PR[90,2] + -7.111;
   1:L PR[91] R[100]mm/sec CNT100;
   1:  PR[91,1] = PR[90,1] + 25.602;
   1:  PR[91,2] = PR[90,2] + -6.711;
   1:L PR[91] R[100]mm/sec CNT100;
   1:  PR[91,1] = PR[90,1] + 25.670;
   1:  PR[91,2] = PR[90,2] + -6.303;
   1:L PR[91] R[100]mm/sec CNT100;
   1:  PR[91,1] = PR[90,1] + 25.705;
   1:  PR[91,2] = PR[90,2] + -5.670;
   1:L PR[91] R[100]mm/sec CNT100;
   1:  PR[91,1] = PR[90,1] + 26.345;
   1:  PR[91,2] = PR[90,2] + -0.402;
   1:L PR[91] R[100]mm/sec CNT100;
   1:  PR[91,1] = PR[90,1] + 26.245;
   1:  PR[91,2] = PR[90,2] + 0.571;
   1:L PR[91] R[100]mm/sec CNT100;
   1:  PR[91,1] = PR[90,1] + 25.611;
   1:  PR[91,2] = PR[90,2] + 5.790;
   1:L PR[91] R[100]mm/sec CNT100;
   1:  PR[91,1] = PR[90,1] + 25.326;
   1:  PR[91,2] = PR[90,2] + 6.690;
   1:L PR[91] R[100]mm/sec CNT100;
   1:  PR[91,1] = PR[90,1] + 23.458;
   1:  PR[91,2] = PR[90,2] + 11.615;
   1:L PR[91] R[100]mm/sec CNT100;
   1:  PR[91,1] = PR[90,1] + 23.030;
   1:  PR[91,2] = PR[90,2] + 12.382;
   1:L PR[91] R[100]mm/sec CNT100;
   1:  PR[91,1] = PR[90,1] + 22.703;
   1:  PR[91,2] = PR[90,2] + 12.798;
   1:L PR[91] R[100]mm/sec CNT100;
   1:  PR[91,1] = PR[90,1] + 19.630;
   1:  PR[91,2] = PR[90,2] + 17.249;
   1:L PR[91] R[100]mm/sec CNT100;
   1:  PR[91,1] = PR[90,1] + 19.405;
   1:  PR[91,2] = PR[90,2] + 17.479;
   1:L PR[91] R[100]mm/sec CNT100;
   1:  PR[91,1] = PR[90,1] + 18.898;
   1:  PR[91,2] = PR[90,2] + 17.887;
   1:L PR[91] R[100]mm/sec CNT100;
   1:  PR[91,1] = PR[90,1] + 14.856;
   1:  PR[91,2] = PR[90,2] + 21.469;
   1:L PR[91] R[100]mm/sec CNT100;
   1:  PR[91,1] = PR[90,1] + 14.530;
   1:  PR[91,2] = PR[90,2] + 21.670;
   1:L PR[91] R[100]mm/sec CNT100;
   1:  PR[91,1] = PR[90,1] + 13.940;
   1:  PR[91,2] = PR[90,2] + 21.942;
   1:L PR[91] R[100]mm/sec CNT100;
   1:  PR[91,1] = PR[90,1] + 9.154;
   1:  PR[91,2] = PR[90,2] + 24.454;
   1:L PR[91] R[100]mm/sec CNT100;
   1:  PR[91,1] = PR[90,1] + 8.795;
   1:  PR[91,2] = PR[90,2] + 24.568;
   1:L PR[91] R[100]mm/sec CNT100;
   1:  PR[91,1] = PR[90,1] + 8.150;
   1:  PR[91,2] = PR[90,2] + 24.688;
   1:L PR[91] R[100]mm/sec CNT100;
   1:  PR[91,1] = PR[90,1] + 2.907;
   1:  PR[91,2] = PR[90,2] + 25.981;
   1:L PR[91] R[100]mm/sec CNT100;
   1:  PR[91,1] = PR[90,1] + 2.463;
   1:  PR[91,2] = PR[90,2] + 26.008;
   1:L PR[91] R[100]mm/sec CNT100 TB   .50sec,CALL END_PUD;
   1:  DO[117:Laser Start]=OFF;
   1:  PR[92] = PR[91];
   1:  PR[92,3] = PR[92,3] + 50;
   1:J PR[92] 10% FINE;
   1:  WAIT   5.00(sec);
   1:  DO[119:Gas]=OFF;
   1:  CALL HOME_ALL;
/POS
/END
